// TIA Portal V19 export
FUNCTION "PREMIXING" : Void   // FC19, LAD
{ S7_Optimized_Access := 'TRUE' }
// stored: SetENOAutomatically false
   VAR_TEMP   // added for the SCL form of the ladder/FBD networks
      _w1 : Bool;
   END_VAR
BEGIN

REGION Network 2: START MFG PROCESS
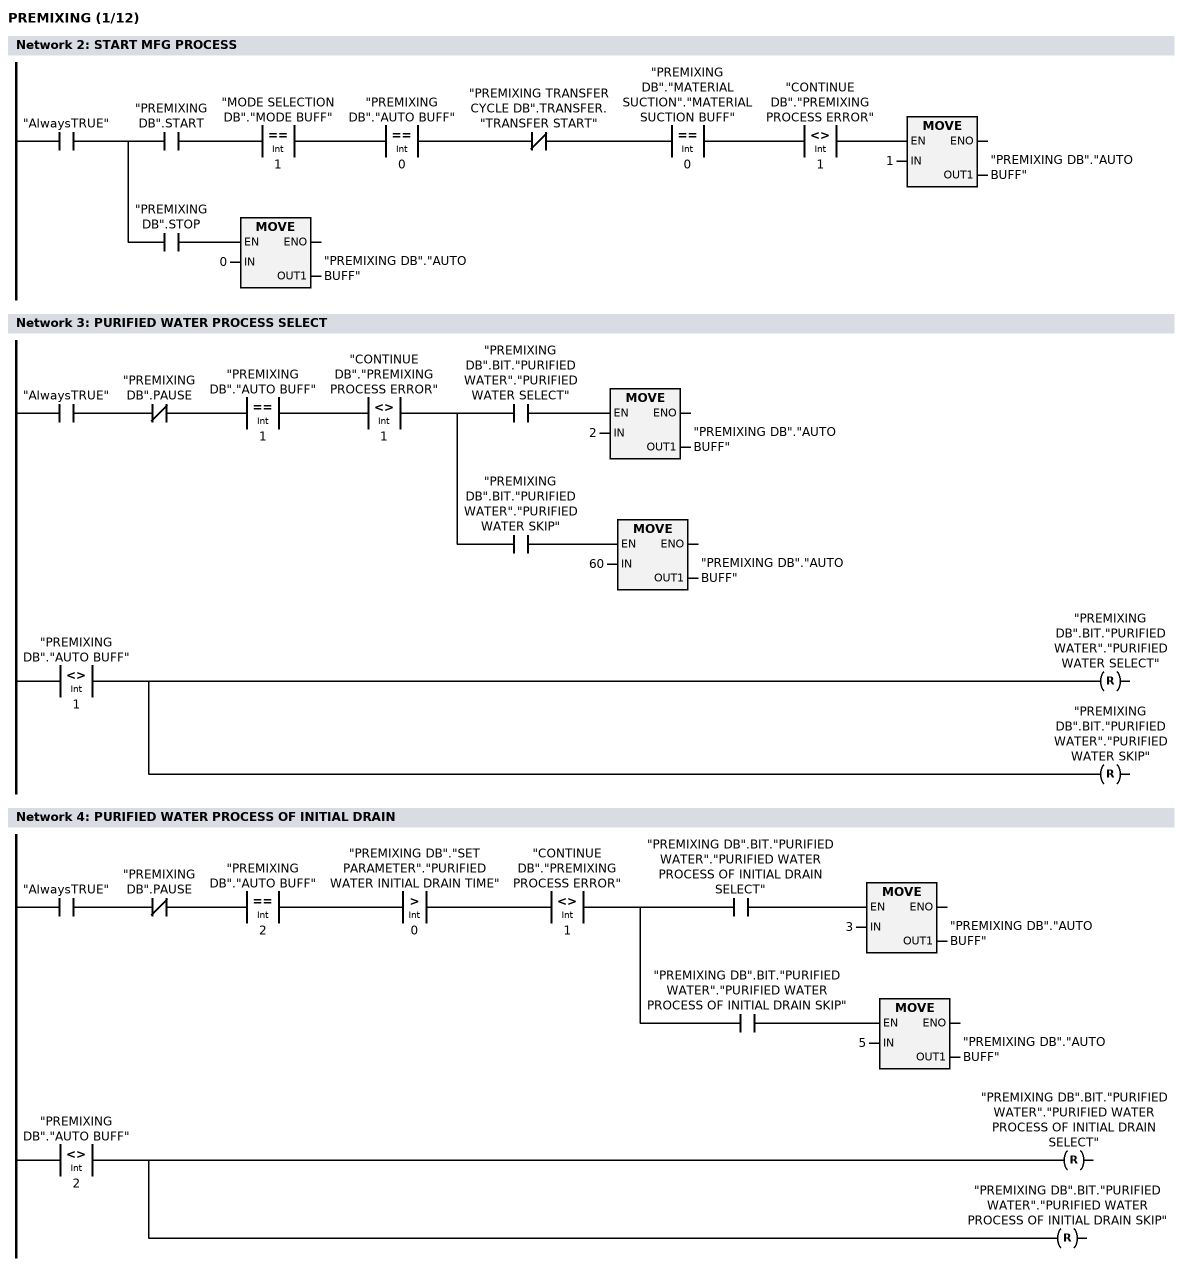
   RUNG wire#powerrail
      Contact( "AlwaysTRUE" )
      wire#w1
      Contact( "PREMIXING DB".START )
      { S7_Templates := "SrcType := Int" } EQ_Contact(in1 := "MODE SELECTION DB"."MODE BUFF", in2 := 1)
      { S7_Templates := "SrcType := Int" } EQ_Contact(in1 := "PREMIXING DB"."AUTO BUFF", in2 := 0)
      I_Contact( "PREMIXING TRANSFER CYCLE DB".TRANSFER."TRANSFER START" )
      { S7_Templates := "SrcType := Int" } EQ_Contact(in1 := "PREMIXING DB"."MATERIAL SUCTION"."MATERIAL SUCTION BUFF", in2 := 0)
      { S7_Templates := "SrcType := Int" } NE_Contact(in1 := "CONTINUE DB"."PREMIXING PROCESS ERROR", in2 := 1)
      Move(in := 1, out1 => "PREMIXING DB"."AUTO BUFF")
   END_RUNG
   RUNG wire#w1
      Contact( "PREMIXING DB".STOP )
      Move(in := 0, out1 => "PREMIXING DB"."AUTO BUFF")
   END_RUNG
   // the same network as SCL:
   IF "AlwaysTRUE" AND "PREMIXING DB".START AND ("MODE SELECTION DB"."MODE BUFF" = 1) AND ("PREMIXING DB"."AUTO BUFF" = 0) AND NOT "PREMIXING TRANSFER CYCLE DB".TRANSFER."TRANSFER START" AND ("PREMIXING DB"."MATERIAL SUCTION"."MATERIAL SUCTION BUFF" = 0) AND ("CONTINUE DB"."PREMIXING PROCESS ERROR" <> 1) THEN
       "PREMIXING DB"."AUTO BUFF" := 1;
   END_IF;
   IF "AlwaysTRUE" AND "PREMIXING DB".STOP THEN "PREMIXING DB"."AUTO BUFF" := 0; END_IF;
END_REGION

REGION Network 3: PURIFIED WATER PROCESS SELECT
   RUNG wire#powerrail
      Contact( "AlwaysTRUE" )
      I_Contact( "PREMIXING DB".PAUSE )
      { S7_Templates := "SrcType := Int" } EQ_Contact(in1 := "PREMIXING DB"."AUTO BUFF", in2 := 1)
      { S7_Templates := "SrcType := Int" } NE_Contact(in1 := "CONTINUE DB"."PREMIXING PROCESS ERROR", in2 := 1)
      wire#w1
      Contact( "PREMIXING DB".BIT."PURIFIED WATER"."PURIFIED WATER SELECT" )
      Move(in := 2, out1 => "PREMIXING DB"."AUTO BUFF")
   END_RUNG
   RUNG wire#w1
      Contact( "PREMIXING DB".BIT."PURIFIED WATER"."PURIFIED WATER SKIP" )
      Move(in := 60, out1 => "PREMIXING DB"."AUTO BUFF")
   END_RUNG
   RUNG wire#powerrail
      { S7_Templates := "SrcType := Int" } NE_Contact(in1 := "PREMIXING DB"."AUTO BUFF", in2 := 1)
      wire#w2
      R_Coil( "PREMIXING DB".BIT."PURIFIED WATER"."PURIFIED WATER SELECT" )
   END_RUNG
   RUNG wire#w2
      R_Coil( "PREMIXING DB".BIT."PURIFIED WATER"."PURIFIED WATER SKIP" )
   END_RUNG
   // the same network as SCL:
   #_w1 := "AlwaysTRUE" AND NOT "PREMIXING DB".PAUSE AND ("PREMIXING DB"."AUTO BUFF" = 1) AND ("CONTINUE DB"."PREMIXING PROCESS ERROR" <> 1);
   IF #_w1 AND "PREMIXING DB".BIT."PURIFIED WATER"."PURIFIED WATER SELECT" THEN
       "PREMIXING DB"."AUTO BUFF" := 2;
   END_IF;
   IF #_w1 AND "PREMIXING DB".BIT."PURIFIED WATER"."PURIFIED WATER SKIP" THEN
       "PREMIXING DB"."AUTO BUFF" := 60;
   END_IF;
   IF "PREMIXING DB"."AUTO BUFF" <> 1 THEN
       "PREMIXING DB".BIT."PURIFIED WATER"."PURIFIED WATER SELECT" := FALSE;
       "PREMIXING DB".BIT."PURIFIED WATER"."PURIFIED WATER SKIP" := FALSE;
   END_IF;
END_REGION

REGION Network 4: PURIFIED WATER PROCESS OF INITIAL DRAIN
   RUNG wire#powerrail
      Contact( "AlwaysTRUE" )
      I_Contact( "PREMIXING DB".PAUSE )
      { S7_Templates := "SrcType := Int" } EQ_Contact(in1 := "PREMIXING DB"."AUTO BUFF", in2 := 2)
      { S7_Templates := "SrcType := Int" } GT_Contact(in1 := "PREMIXING DB"."SET PARAMETER"."PURIFIED WATER INITIAL DRAIN TIME", in2 := 0)
      { S7_Templates := "SrcType := Int" } NE_Contact(in1 := "CONTINUE DB"."PREMIXING PROCESS ERROR", in2 := 1)
      wire#w1
      Contact( "PREMIXING DB".BIT."PURIFIED WATER"."PURIFIED WATER PROCESS OF INITIAL DRAIN SELECT" )
      Move(in := 3, out1 => "PREMIXING DB"."AUTO BUFF")
   END_RUNG
   RUNG wire#w1
      Contact( "PREMIXING DB".BIT."PURIFIED WATER"."PURIFIED WATER PROCESS OF INITIAL DRAIN SKIP" )
      Move(in := 5, out1 => "PREMIXING DB"."AUTO BUFF")
   END_RUNG
   RUNG wire#powerrail
      { S7_Templates := "SrcType := Int" } NE_Contact(in1 := "PREMIXING DB"."AUTO BUFF", in2 := 2)
      wire#w2
      R_Coil( "PREMIXING DB".BIT."PURIFIED WATER"."PURIFIED WATER PROCESS OF INITIAL DRAIN SELECT" )
   END_RUNG
   RUNG wire#w2
      R_Coil( "PREMIXING DB".BIT."PURIFIED WATER"."PURIFIED WATER PROCESS OF INITIAL DRAIN SKIP" )
   END_RUNG
   // the same network as SCL:
   #_w1 := "AlwaysTRUE" AND NOT "PREMIXING DB".PAUSE AND ("PREMIXING DB"."AUTO BUFF" = 2) AND ("PREMIXING DB"."SET PARAMETER"."PURIFIED WATER INITIAL DRAIN TIME" > 0) AND ("CONTINUE DB"."PREMIXING PROCESS ERROR" <> 1);
   IF #_w1 AND "PREMIXING DB".BIT."PURIFIED WATER"."PURIFIED WATER PROCESS OF INITIAL DRAIN SELECT" THEN
       "PREMIXING DB"."AUTO BUFF" := 3;
   END_IF;
   IF #_w1 AND "PREMIXING DB".BIT."PURIFIED WATER"."PURIFIED WATER PROCESS OF INITIAL DRAIN SKIP" THEN
       "PREMIXING DB"."AUTO BUFF" := 5;
   END_IF;
   IF "PREMIXING DB"."AUTO BUFF" <> 2 THEN
       "PREMIXING DB".BIT."PURIFIED WATER"."PURIFIED WATER PROCESS OF INITIAL DRAIN SELECT" := FALSE;
       "PREMIXING DB".BIT."PURIFIED WATER"."PURIFIED WATER PROCESS OF INITIAL DRAIN SKIP" := FALSE;
   END_IF;
END_REGION

REGION Network 5: TIMER
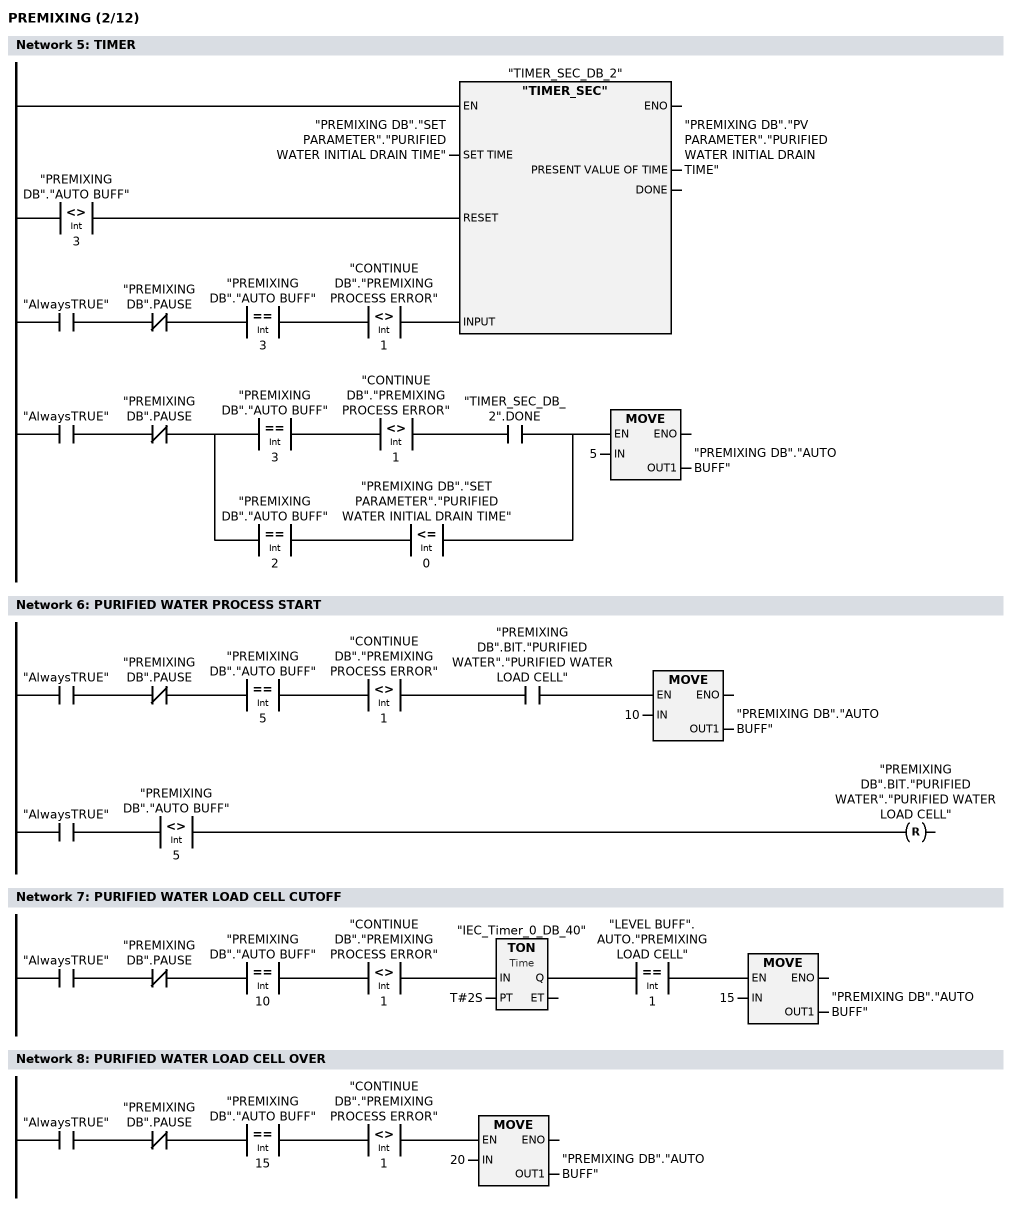
   RUNG wire#powerrail
      "TIMER_SEC_DB_2"(RESET := wire#w1, INPUT := wire#w2, "SET TIME" := "PREMIXING DB"."SET PARAMETER"."PURIFIED WATER INITIAL DRAIN TIME", "PRESENT VALUE OF TIME" => "PREMIXING DB"."PV PARAMETER"."PURIFIED WATER INITIAL DRAIN TIME", DONE =>)
   END_RUNG
   RUNG wire#powerrail
      { S7_Templates := "SrcType := Int" } NE_Contact(in1 := "PREMIXING DB"."AUTO BUFF", in2 := 3)
   END_RUNG wire#w1
   RUNG wire#powerrail
      Contact( "AlwaysTRUE" )
      I_Contact( "PREMIXING DB".PAUSE )
      { S7_Templates := "SrcType := Int" } EQ_Contact(in1 := "PREMIXING DB"."AUTO BUFF", in2 := 3)
      { S7_Templates := "SrcType := Int" } NE_Contact(in1 := "CONTINUE DB"."PREMIXING PROCESS ERROR", in2 := 1)
   END_RUNG wire#w2
   RUNG wire#powerrail
      Contact( "AlwaysTRUE" )
      I_Contact( "PREMIXING DB".PAUSE )
      wire#w3
      { S7_Templates := "SrcType := Int" } EQ_Contact(in1 := "PREMIXING DB"."AUTO BUFF", in2 := 3)
      { S7_Templates := "SrcType := Int" } NE_Contact(in1 := "CONTINUE DB"."PREMIXING PROCESS ERROR", in2 := 1)
      Contact( "TIMER_SEC_DB_2".DONE )
      wire#w4
      Move(in := 5, out1 => "PREMIXING DB"."AUTO BUFF")
   END_RUNG
   RUNG wire#w3
      { S7_Templates := "SrcType := Int" } EQ_Contact(in1 := "PREMIXING DB"."AUTO BUFF", in2 := 2)
      { S7_Templates := "SrcType := Int" } LE_Contact(in1 := "PREMIXING DB"."SET PARAMETER"."PURIFIED WATER INITIAL DRAIN TIME", in2 := 0)
   END_RUNG wire#w4
   // the same network as SCL:
   "TIMER_SEC_DB_2"("SET TIME" := "PREMIXING DB"."SET PARAMETER"."PURIFIED WATER INITIAL DRAIN TIME",   // "TIMER_SEC"
                    RESET := "PREMIXING DB"."AUTO BUFF" <> 3,
                    INPUT := "AlwaysTRUE" AND NOT "PREMIXING DB".PAUSE AND ("PREMIXING DB"."AUTO BUFF" = 3) AND ("CONTINUE DB"."PREMIXING PROCESS ERROR" <> 1),
                    "PRESENT VALUE OF TIME" => "PREMIXING DB"."PV PARAMETER"."PURIFIED WATER INITIAL DRAIN TIME");
   IF "AlwaysTRUE" AND NOT "PREMIXING DB".PAUSE AND ((("PREMIXING DB"."AUTO BUFF" = 3) AND ("CONTINUE DB"."PREMIXING PROCESS ERROR" <> 1) AND "TIMER_SEC_DB_2".DONE) OR (("PREMIXING DB"."AUTO BUFF" = 2) AND ("PREMIXING DB"."SET PARAMETER"."PURIFIED WATER INITIAL DRAIN TIME" <= 0))) THEN
       "PREMIXING DB"."AUTO BUFF" := 5;
   END_IF;
END_REGION

REGION Network 6: PURIFIED WATER PROCESS START
   RUNG wire#powerrail
      Contact( "AlwaysTRUE" )
      I_Contact( "PREMIXING DB".PAUSE )
      { S7_Templates := "SrcType := Int" } EQ_Contact(in1 := "PREMIXING DB"."AUTO BUFF", in2 := 5)
      { S7_Templates := "SrcType := Int" } NE_Contact(in1 := "CONTINUE DB"."PREMIXING PROCESS ERROR", in2 := 1)
      Contact( "PREMIXING DB".BIT."PURIFIED WATER"."PURIFIED WATER LOAD CELL" )
      Move(in := 10, out1 => "PREMIXING DB"."AUTO BUFF")
   END_RUNG
   RUNG wire#powerrail
      Contact( "AlwaysTRUE" )
      { S7_Templates := "SrcType := Int" } NE_Contact(in1 := "PREMIXING DB"."AUTO BUFF", in2 := 5)
      R_Coil( "PREMIXING DB".BIT."PURIFIED WATER"."PURIFIED WATER LOAD CELL" )
   END_RUNG
   // the same network as SCL:
   IF "AlwaysTRUE" AND NOT "PREMIXING DB".PAUSE AND ("PREMIXING DB"."AUTO BUFF" = 5) AND ("CONTINUE DB"."PREMIXING PROCESS ERROR" <> 1) AND "PREMIXING DB".BIT."PURIFIED WATER"."PURIFIED WATER LOAD CELL" THEN
       "PREMIXING DB"."AUTO BUFF" := 10;
   END_IF;
   IF "AlwaysTRUE" AND ("PREMIXING DB"."AUTO BUFF" <> 5) THEN
       "PREMIXING DB".BIT."PURIFIED WATER"."PURIFIED WATER LOAD CELL" := FALSE;
   END_IF;
END_REGION

REGION Network 7: PURIFIED WATER LOAD CELL CUTOFF
   RUNG wire#powerrail
      Contact( "AlwaysTRUE" )
      I_Contact( "PREMIXING DB".PAUSE )
      { S7_Templates := "SrcType := Int" } EQ_Contact(in1 := "PREMIXING DB"."AUTO BUFF", in2 := 10)
      { S7_Templates := "SrcType := Int" } NE_Contact(in1 := "CONTINUE DB"."PREMIXING PROCESS ERROR", in2 := 1)
      { S7_Templates := "time_type := Time" } "IEC_Timer_0_DB_40".TON(pt := T#2S, et =>)
      { S7_Templates := "SrcType := Int" } EQ_Contact(in1 := "LEVEL BUFF".AUTO."PREMIXING LOAD CELL", in2 := 1)
      Move(in := 15, out1 => "PREMIXING DB"."AUTO BUFF")
   END_RUNG
   // the same network as SCL:
   "IEC_Timer_0_DB_40".TON(IN := "AlwaysTRUE" AND NOT "PREMIXING DB".PAUSE AND ("PREMIXING DB"."AUTO BUFF" = 10) AND ("CONTINUE DB"."PREMIXING PROCESS ERROR" <> 1),
                           PT := T#2S);
   IF "IEC_Timer_0_DB_40".Q AND ("LEVEL BUFF".AUTO."PREMIXING LOAD CELL" = 1) THEN
       "PREMIXING DB"."AUTO BUFF" := 15;
   END_IF;
END_REGION

REGION Network 8: PURIFIED WATER LOAD CELL OVER
   RUNG wire#powerrail
      Contact( "AlwaysTRUE" )
      I_Contact( "PREMIXING DB".PAUSE )
      { S7_Templates := "SrcType := Int" } EQ_Contact(in1 := "PREMIXING DB"."AUTO BUFF", in2 := 15)
      { S7_Templates := "SrcType := Int" } NE_Contact(in1 := "CONTINUE DB"."PREMIXING PROCESS ERROR", in2 := 1)
      Move(in := 20, out1 => "PREMIXING DB"."AUTO BUFF")
   END_RUNG
   // the same network as SCL:
   IF "AlwaysTRUE" AND NOT "PREMIXING DB".PAUSE AND ("PREMIXING DB"."AUTO BUFF" = 15) AND ("CONTINUE DB"."PREMIXING PROCESS ERROR" <> 1) THEN
       "PREMIXING DB"."AUTO BUFF" := 20;
   END_IF;
END_REGION

REGION Network 9: PURIFIED WATER HEATING OR COOLING SEL
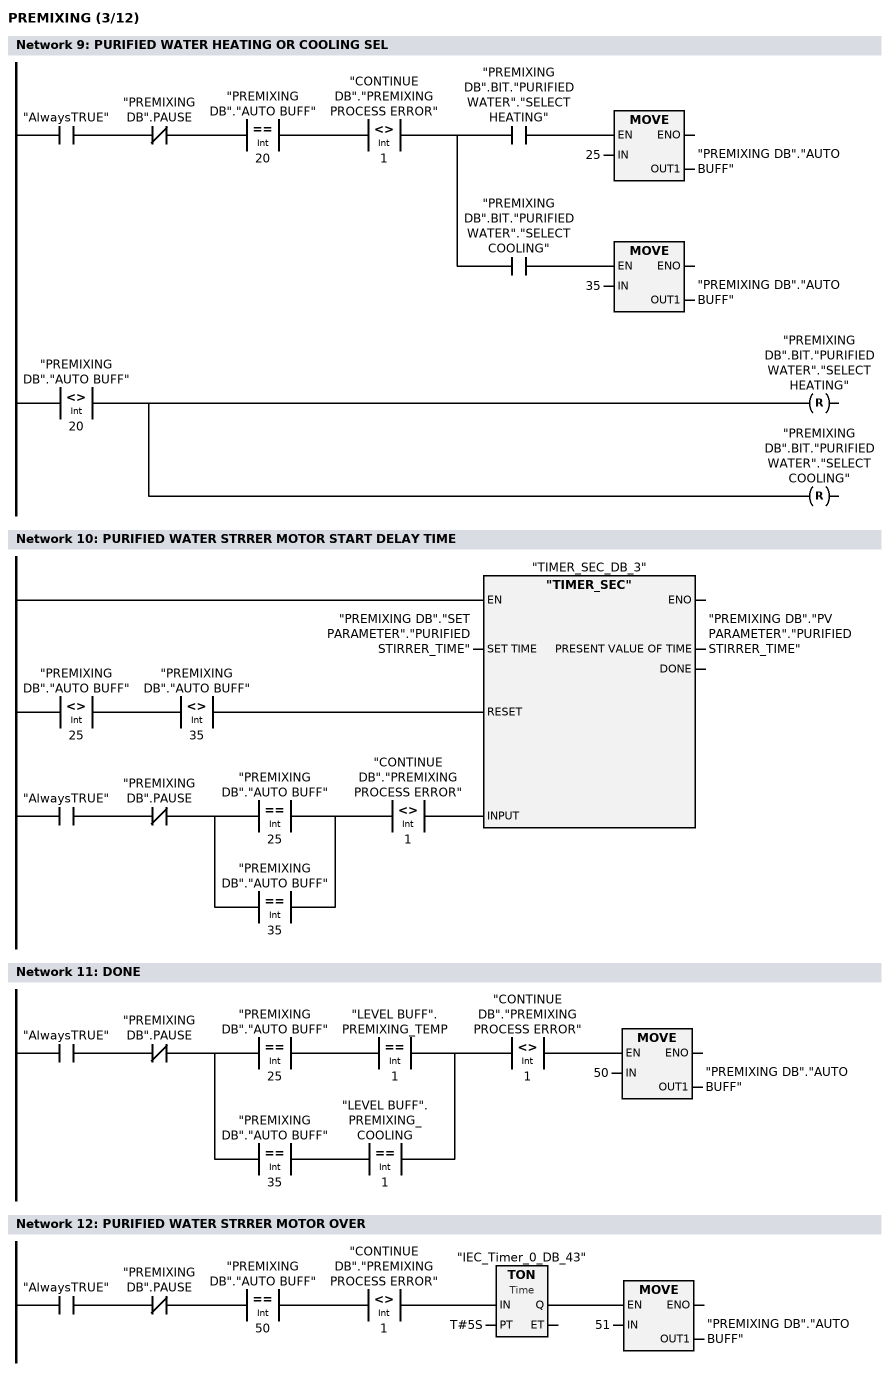
   RUNG wire#powerrail
      Contact( "AlwaysTRUE" )
      I_Contact( "PREMIXING DB".PAUSE )
      { S7_Templates := "SrcType := Int" } EQ_Contact(in1 := "PREMIXING DB"."AUTO BUFF", in2 := 20)
      { S7_Templates := "SrcType := Int" } NE_Contact(in1 := "CONTINUE DB"."PREMIXING PROCESS ERROR", in2 := 1)
      wire#w1
      Contact( "PREMIXING DB".BIT."PURIFIED WATER"."SELECT HEATING" )
      Move(in := 25, out1 => "PREMIXING DB"."AUTO BUFF")
   END_RUNG
   RUNG wire#w1
      Contact( "PREMIXING DB".BIT."PURIFIED WATER"."SELECT COOLING" )
      Move(in := 35, out1 => "PREMIXING DB"."AUTO BUFF")
   END_RUNG
   RUNG wire#powerrail
      { S7_Templates := "SrcType := Int" } NE_Contact(in1 := "PREMIXING DB"."AUTO BUFF", in2 := 20)
      wire#w2
      R_Coil( "PREMIXING DB".BIT."PURIFIED WATER"."SELECT HEATING" )
   END_RUNG
   RUNG wire#w2
      R_Coil( "PREMIXING DB".BIT."PURIFIED WATER"."SELECT COOLING" )
   END_RUNG
   // the same network as SCL:
   #_w1 := "AlwaysTRUE" AND NOT "PREMIXING DB".PAUSE AND ("PREMIXING DB"."AUTO BUFF" = 20) AND ("CONTINUE DB"."PREMIXING PROCESS ERROR" <> 1);
   IF #_w1 AND "PREMIXING DB".BIT."PURIFIED WATER"."SELECT HEATING" THEN
       "PREMIXING DB"."AUTO BUFF" := 25;
   END_IF;
   IF #_w1 AND "PREMIXING DB".BIT."PURIFIED WATER"."SELECT COOLING" THEN
       "PREMIXING DB"."AUTO BUFF" := 35;
   END_IF;
   IF "PREMIXING DB"."AUTO BUFF" <> 20 THEN
       "PREMIXING DB".BIT."PURIFIED WATER"."SELECT HEATING" := FALSE;
       "PREMIXING DB".BIT."PURIFIED WATER"."SELECT COOLING" := FALSE;
   END_IF;
END_REGION

REGION Network 10: PURIFIED WATER STRRER MOTOR START DELAY TIME
   RUNG wire#powerrail
      "TIMER_SEC_DB_3"(RESET := wire#w1, INPUT := wire#w4, "SET TIME" := "PREMIXING DB"."SET PARAMETER"."PURIFIED STIRRER_TIME", "PRESENT VALUE OF TIME" => "PREMIXING DB"."PV PARAMETER"."PURIFIED STIRRER_TIME", DONE =>)
   END_RUNG
   RUNG wire#powerrail
      { S7_Templates := "SrcType := Int" } NE_Contact(in1 := "PREMIXING DB"."AUTO BUFF", in2 := 25)
      { S7_Templates := "SrcType := Int" } NE_Contact(in1 := "PREMIXING DB"."AUTO BUFF", in2 := 35)
   END_RUNG wire#w1
   RUNG wire#powerrail
      Contact( "AlwaysTRUE" )
      I_Contact( "PREMIXING DB".PAUSE )
      wire#w2
      { S7_Templates := "SrcType := Int" } EQ_Contact(in1 := "PREMIXING DB"."AUTO BUFF", in2 := 25)
      wire#w3
      { S7_Templates := "SrcType := Int" } NE_Contact(in1 := "CONTINUE DB"."PREMIXING PROCESS ERROR", in2 := 1)
   END_RUNG wire#w4
   RUNG wire#w2
      { S7_Templates := "SrcType := Int" } EQ_Contact(in1 := "PREMIXING DB"."AUTO BUFF", in2 := 35)
   END_RUNG wire#w3
   // the same network as SCL:
   "TIMER_SEC_DB_3"("SET TIME" := "PREMIXING DB"."SET PARAMETER"."PURIFIED STIRRER_TIME",   // "TIMER_SEC"
                    RESET := ("PREMIXING DB"."AUTO BUFF" <> 25) AND ("PREMIXING DB"."AUTO BUFF" <> 35),
                    INPUT := "AlwaysTRUE" AND NOT "PREMIXING DB".PAUSE AND (("PREMIXING DB"."AUTO BUFF" = 25) OR ("PREMIXING DB"."AUTO BUFF" = 35)) AND ("CONTINUE DB"."PREMIXING PROCESS ERROR" <> 1),
                    "PRESENT VALUE OF TIME" => "PREMIXING DB"."PV PARAMETER"."PURIFIED STIRRER_TIME");
END_REGION

REGION Network 11: DONE
   RUNG wire#powerrail
      Contact( "AlwaysTRUE" )
      I_Contact( "PREMIXING DB".PAUSE )
      wire#w1
      { S7_Templates := "SrcType := Int" } EQ_Contact(in1 := "PREMIXING DB"."AUTO BUFF", in2 := 25)
      { S7_Templates := "SrcType := Int" } EQ_Contact(in1 := "LEVEL BUFF".PREMIXING_TEMP, in2 := 1)
      wire#w2
      { S7_Templates := "SrcType := Int" } NE_Contact(in1 := "CONTINUE DB"."PREMIXING PROCESS ERROR", in2 := 1)
      Move(in := 50, out1 => "PREMIXING DB"."AUTO BUFF")
   END_RUNG
   RUNG wire#w1
      { S7_Templates := "SrcType := Int" } EQ_Contact(in1 := "PREMIXING DB"."AUTO BUFF", in2 := 35)
      { S7_Templates := "SrcType := Int" } EQ_Contact(in1 := "LEVEL BUFF".PREMIXING_COOLING, in2 := 1)
   END_RUNG wire#w2
   // the same network as SCL:
   IF "AlwaysTRUE" AND NOT "PREMIXING DB".PAUSE AND ((("PREMIXING DB"."AUTO BUFF" = 25) AND ("LEVEL BUFF".PREMIXING_TEMP = 1)) OR (("PREMIXING DB"."AUTO BUFF" = 35) AND ("LEVEL BUFF".PREMIXING_COOLING = 1))) AND ("CONTINUE DB"."PREMIXING PROCESS ERROR" <> 1) THEN
       "PREMIXING DB"."AUTO BUFF" := 50;
   END_IF;
END_REGION

REGION Network 12: PURIFIED WATER STRRER MOTOR OVER
   RUNG wire#powerrail
      Contact( "AlwaysTRUE" )
      I_Contact( "PREMIXING DB".PAUSE )
      { S7_Templates := "SrcType := Int" } EQ_Contact(in1 := "PREMIXING DB"."AUTO BUFF", in2 := 50)
      { S7_Templates := "SrcType := Int" } NE_Contact(in1 := "CONTINUE DB"."PREMIXING PROCESS ERROR", in2 := 1)
      { S7_Templates := "time_type := Time" } "IEC_Timer_0_DB_43".TON(pt := T#5S, et =>)
      Move(in := 51, out1 => "PREMIXING DB"."AUTO BUFF")
   END_RUNG
   // the same network as SCL:
   "IEC_Timer_0_DB_43".TON(IN := "AlwaysTRUE" AND NOT "PREMIXING DB".PAUSE AND ("PREMIXING DB"."AUTO BUFF" = 50) AND ("CONTINUE DB"."PREMIXING PROCESS ERROR" <> 1),
                           PT := T#5S);
   IF "IEC_Timer_0_DB_43".Q THEN "PREMIXING DB"."AUTO BUFF" := 51; END_IF;
END_REGION

REGION Network 13: PURIFIED WATER PROCESS OF JACKET DRAIN
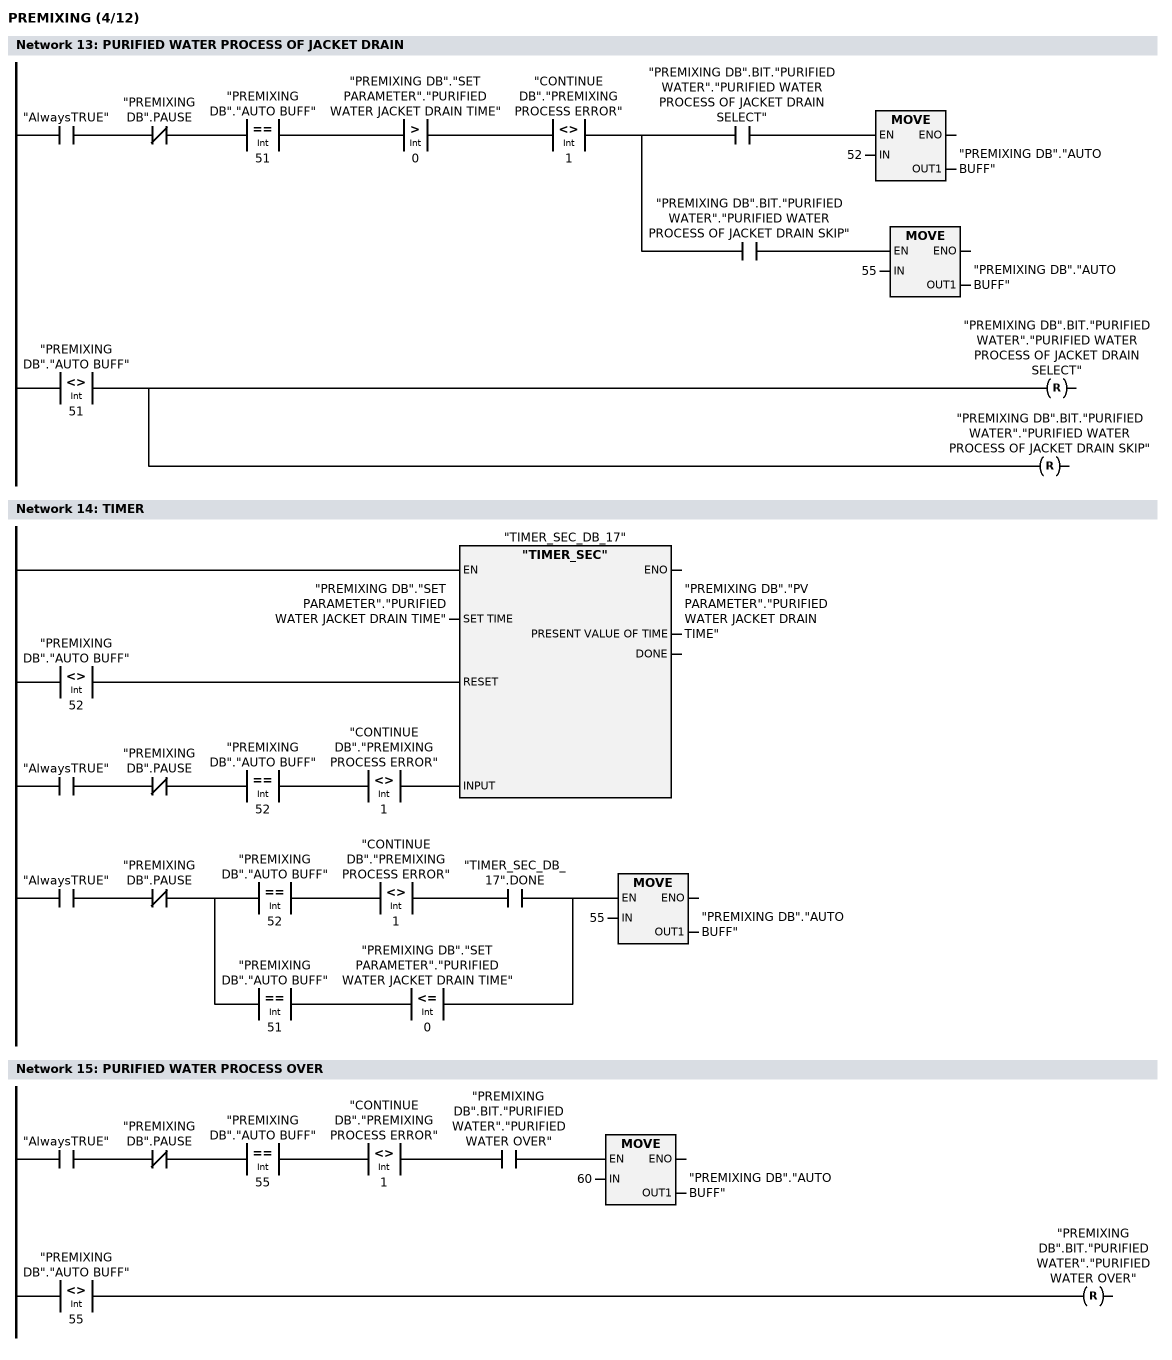
   RUNG wire#powerrail
      Contact( "AlwaysTRUE" )
      I_Contact( "PREMIXING DB".PAUSE )
      { S7_Templates := "SrcType := Int" } EQ_Contact(in1 := "PREMIXING DB"."AUTO BUFF", in2 := 51)
      { S7_Templates := "SrcType := Int" } GT_Contact(in1 := "PREMIXING DB"."SET PARAMETER"."PURIFIED WATER JACKET DRAIN TIME", in2 := 0)
      { S7_Templates := "SrcType := Int" } NE_Contact(in1 := "CONTINUE DB"."PREMIXING PROCESS ERROR", in2 := 1)
      wire#w1
      Contact( "PREMIXING DB".BIT."PURIFIED WATER"."PURIFIED WATER PROCESS OF JACKET DRAIN SELECT" )
      Move(in := 52, out1 => "PREMIXING DB"."AUTO BUFF")
   END_RUNG
   RUNG wire#w1
      Contact( "PREMIXING DB".BIT."PURIFIED WATER"."PURIFIED WATER PROCESS OF JACKET DRAIN SKIP" )
      Move(in := 55, out1 => "PREMIXING DB"."AUTO BUFF")
   END_RUNG
   RUNG wire#powerrail
      { S7_Templates := "SrcType := Int" } NE_Contact(in1 := "PREMIXING DB"."AUTO BUFF", in2 := 51)
      wire#w2
      R_Coil( "PREMIXING DB".BIT."PURIFIED WATER"."PURIFIED WATER PROCESS OF JACKET DRAIN SELECT" )
   END_RUNG
   RUNG wire#w2
      R_Coil( "PREMIXING DB".BIT."PURIFIED WATER"."PURIFIED WATER PROCESS OF JACKET DRAIN SKIP" )
   END_RUNG
   // the same network as SCL:
   #_w1 := "AlwaysTRUE" AND NOT "PREMIXING DB".PAUSE AND ("PREMIXING DB"."AUTO BUFF" = 51) AND ("PREMIXING DB"."SET PARAMETER"."PURIFIED WATER JACKET DRAIN TIME" > 0) AND ("CONTINUE DB"."PREMIXING PROCESS ERROR" <> 1);
   IF #_w1 AND "PREMIXING DB".BIT."PURIFIED WATER"."PURIFIED WATER PROCESS OF JACKET DRAIN SELECT" THEN
       "PREMIXING DB"."AUTO BUFF" := 52;
   END_IF;
   IF #_w1 AND "PREMIXING DB".BIT."PURIFIED WATER"."PURIFIED WATER PROCESS OF JACKET DRAIN SKIP" THEN
       "PREMIXING DB"."AUTO BUFF" := 55;
   END_IF;
   IF "PREMIXING DB"."AUTO BUFF" <> 51 THEN
       "PREMIXING DB".BIT."PURIFIED WATER"."PURIFIED WATER PROCESS OF JACKET DRAIN SELECT" := FALSE;
       "PREMIXING DB".BIT."PURIFIED WATER"."PURIFIED WATER PROCESS OF JACKET DRAIN SKIP" := FALSE;
   END_IF;
END_REGION

REGION Network 14: TIMER
   RUNG wire#powerrail
      "TIMER_SEC_DB_17"(RESET := wire#w1, INPUT := wire#w2, "SET TIME" := "PREMIXING DB"."SET PARAMETER"."PURIFIED WATER JACKET DRAIN TIME", "PRESENT VALUE OF TIME" => "PREMIXING DB"."PV PARAMETER"."PURIFIED WATER JACKET DRAIN TIME", DONE =>)
   END_RUNG
   RUNG wire#powerrail
      { S7_Templates := "SrcType := Int" } NE_Contact(in1 := "PREMIXING DB"."AUTO BUFF", in2 := 52)
   END_RUNG wire#w1
   RUNG wire#powerrail
      Contact( "AlwaysTRUE" )
      I_Contact( "PREMIXING DB".PAUSE )
      { S7_Templates := "SrcType := Int" } EQ_Contact(in1 := "PREMIXING DB"."AUTO BUFF", in2 := 52)
      { S7_Templates := "SrcType := Int" } NE_Contact(in1 := "CONTINUE DB"."PREMIXING PROCESS ERROR", in2 := 1)
   END_RUNG wire#w2
   RUNG wire#powerrail
      Contact( "AlwaysTRUE" )
      I_Contact( "PREMIXING DB".PAUSE )
      wire#w3
      { S7_Templates := "SrcType := Int" } EQ_Contact(in1 := "PREMIXING DB"."AUTO BUFF", in2 := 52)
      { S7_Templates := "SrcType := Int" } NE_Contact(in1 := "CONTINUE DB"."PREMIXING PROCESS ERROR", in2 := 1)
      Contact( "TIMER_SEC_DB_17".DONE )
      wire#w4
      Move(in := 55, out1 => "PREMIXING DB"."AUTO BUFF")
   END_RUNG
   RUNG wire#w3
      { S7_Templates := "SrcType := Int" } EQ_Contact(in1 := "PREMIXING DB"."AUTO BUFF", in2 := 51)
      { S7_Templates := "SrcType := Int" } LE_Contact(in1 := "PREMIXING DB"."SET PARAMETER"."PURIFIED WATER JACKET DRAIN TIME", in2 := 0)
   END_RUNG wire#w4
   // the same network as SCL:
   "TIMER_SEC_DB_17"("SET TIME" := "PREMIXING DB"."SET PARAMETER"."PURIFIED WATER JACKET DRAIN TIME",   // "TIMER_SEC"
                     RESET := "PREMIXING DB"."AUTO BUFF" <> 52,
                     INPUT := "AlwaysTRUE" AND NOT "PREMIXING DB".PAUSE AND ("PREMIXING DB"."AUTO BUFF" = 52) AND ("CONTINUE DB"."PREMIXING PROCESS ERROR" <> 1),
                     "PRESENT VALUE OF TIME" => "PREMIXING DB"."PV PARAMETER"."PURIFIED WATER JACKET DRAIN TIME");
   IF "AlwaysTRUE" AND NOT "PREMIXING DB".PAUSE AND ((("PREMIXING DB"."AUTO BUFF" = 52) AND ("CONTINUE DB"."PREMIXING PROCESS ERROR" <> 1) AND "TIMER_SEC_DB_17".DONE) OR (("PREMIXING DB"."AUTO BUFF" = 51) AND ("PREMIXING DB"."SET PARAMETER"."PURIFIED WATER JACKET DRAIN TIME" <= 0))) THEN
       "PREMIXING DB"."AUTO BUFF" := 55;
   END_IF;
END_REGION

REGION Network 15: PURIFIED WATER PROCESS OVER
   RUNG wire#powerrail
      Contact( "AlwaysTRUE" )
      I_Contact( "PREMIXING DB".PAUSE )
      { S7_Templates := "SrcType := Int" } EQ_Contact(in1 := "PREMIXING DB"."AUTO BUFF", in2 := 55)
      { S7_Templates := "SrcType := Int" } NE_Contact(in1 := "CONTINUE DB"."PREMIXING PROCESS ERROR", in2 := 1)
      Contact( "PREMIXING DB".BIT."PURIFIED WATER"."PURIFIED WATER OVER" )
      Move(in := 60, out1 => "PREMIXING DB"."AUTO BUFF")
   END_RUNG
   RUNG wire#powerrail
      { S7_Templates := "SrcType := Int" } NE_Contact(in1 := "PREMIXING DB"."AUTO BUFF", in2 := 55)
      R_Coil( "PREMIXING DB".BIT."PURIFIED WATER"."PURIFIED WATER OVER" )
   END_RUNG
   // the same network as SCL:
   IF "AlwaysTRUE" AND NOT "PREMIXING DB".PAUSE AND ("PREMIXING DB"."AUTO BUFF" = 55) AND ("CONTINUE DB"."PREMIXING PROCESS ERROR" <> 1) AND "PREMIXING DB".BIT."PURIFIED WATER"."PURIFIED WATER OVER" THEN
       "PREMIXING DB"."AUTO BUFF" := 60;
   END_IF;
   IF "PREMIXING DB"."AUTO BUFF" <> 55 THEN
       "PREMIXING DB".BIT."PURIFIED WATER"."PURIFIED WATER OVER" := FALSE;
   END_IF;
END_REGION

REGION Network 17: MATERIAL ADDITION PROCESS SELECT
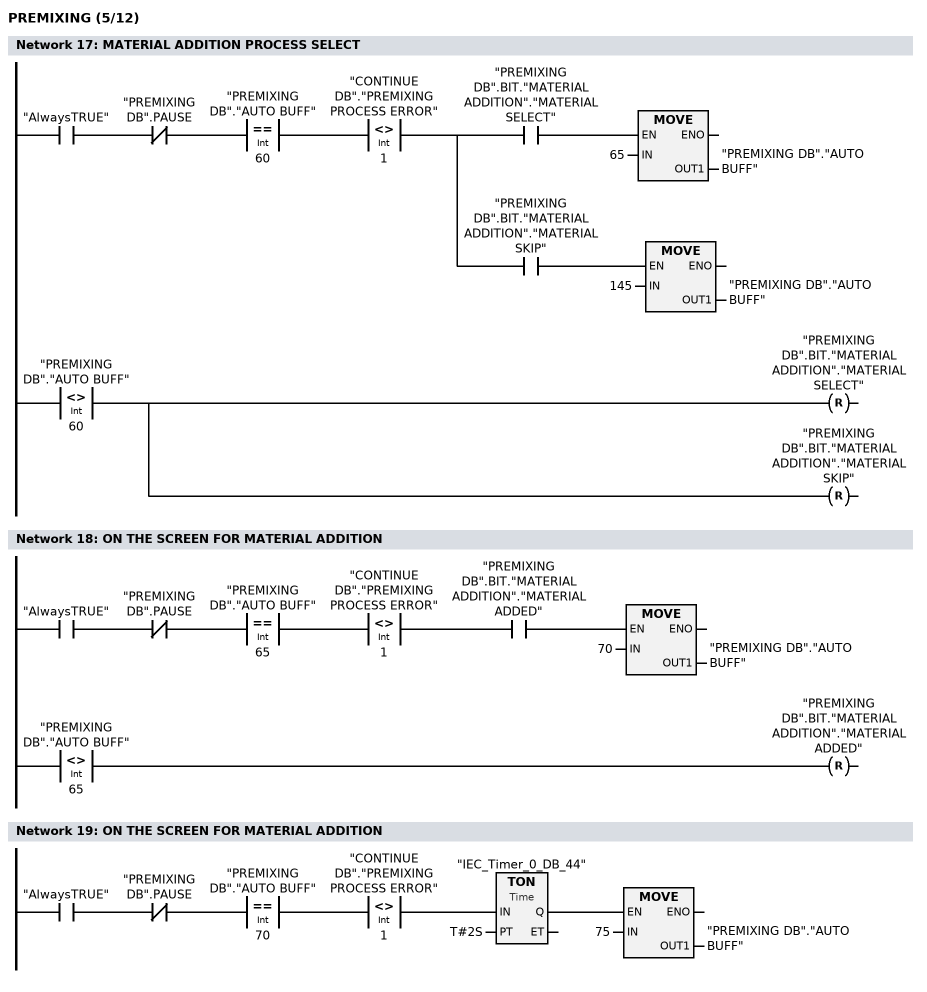
   RUNG wire#powerrail
      Contact( "AlwaysTRUE" )
      I_Contact( "PREMIXING DB".PAUSE )
      { S7_Templates := "SrcType := Int" } EQ_Contact(in1 := "PREMIXING DB"."AUTO BUFF", in2 := 60)
      { S7_Templates := "SrcType := Int" } NE_Contact(in1 := "CONTINUE DB"."PREMIXING PROCESS ERROR", in2 := 1)
      wire#w1
      Contact( "PREMIXING DB".BIT."MATERIAL ADDITION"."MATERIAL SELECT" )
      Move(in := 65, out1 => "PREMIXING DB"."AUTO BUFF")
   END_RUNG
   RUNG wire#w1
      Contact( "PREMIXING DB".BIT."MATERIAL ADDITION"."MATERIAL SKIP" )
      Move(in := 145, out1 => "PREMIXING DB"."AUTO BUFF")
   END_RUNG
   RUNG wire#powerrail
      { S7_Templates := "SrcType := Int" } NE_Contact(in1 := "PREMIXING DB"."AUTO BUFF", in2 := 60)
      wire#w2
      R_Coil( "PREMIXING DB".BIT."MATERIAL ADDITION"."MATERIAL SELECT" )
   END_RUNG
   RUNG wire#w2
      R_Coil( "PREMIXING DB".BIT."MATERIAL ADDITION"."MATERIAL SKIP" )
   END_RUNG
   // the same network as SCL:
   #_w1 := "AlwaysTRUE" AND NOT "PREMIXING DB".PAUSE AND ("PREMIXING DB"."AUTO BUFF" = 60) AND ("CONTINUE DB"."PREMIXING PROCESS ERROR" <> 1);
   IF #_w1 AND "PREMIXING DB".BIT."MATERIAL ADDITION"."MATERIAL SELECT" THEN
       "PREMIXING DB"."AUTO BUFF" := 65;
   END_IF;
   IF #_w1 AND "PREMIXING DB".BIT."MATERIAL ADDITION"."MATERIAL SKIP" THEN
       "PREMIXING DB"."AUTO BUFF" := 145;
   END_IF;
   IF "PREMIXING DB"."AUTO BUFF" <> 60 THEN
       "PREMIXING DB".BIT."MATERIAL ADDITION"."MATERIAL SELECT" := FALSE;
       "PREMIXING DB".BIT."MATERIAL ADDITION"."MATERIAL SKIP" := FALSE;
   END_IF;
END_REGION

REGION Network 18: ON THE SCREEN FOR MATERIAL ADDITION
   RUNG wire#powerrail
      Contact( "AlwaysTRUE" )
      I_Contact( "PREMIXING DB".PAUSE )
      { S7_Templates := "SrcType := Int" } EQ_Contact(in1 := "PREMIXING DB"."AUTO BUFF", in2 := 65)
      { S7_Templates := "SrcType := Int" } NE_Contact(in1 := "CONTINUE DB"."PREMIXING PROCESS ERROR", in2 := 1)
      Contact( "PREMIXING DB".BIT."MATERIAL ADDITION"."MATERIAL ADDED" )
      Move(in := 70, out1 => "PREMIXING DB"."AUTO BUFF")
   END_RUNG
   RUNG wire#powerrail
      { S7_Templates := "SrcType := Int" } NE_Contact(in1 := "PREMIXING DB"."AUTO BUFF", in2 := 65)
      R_Coil( "PREMIXING DB".BIT."MATERIAL ADDITION"."MATERIAL ADDED" )
   END_RUNG
   // the same network as SCL:
   IF "AlwaysTRUE" AND NOT "PREMIXING DB".PAUSE AND ("PREMIXING DB"."AUTO BUFF" = 65) AND ("CONTINUE DB"."PREMIXING PROCESS ERROR" <> 1) AND "PREMIXING DB".BIT."MATERIAL ADDITION"."MATERIAL ADDED" THEN
       "PREMIXING DB"."AUTO BUFF" := 70;
   END_IF;
   IF "PREMIXING DB"."AUTO BUFF" <> 65 THEN
       "PREMIXING DB".BIT."MATERIAL ADDITION"."MATERIAL ADDED" := FALSE;
   END_IF;
END_REGION

REGION Network 19: ON THE SCREEN FOR MATERIAL ADDITION
   RUNG wire#powerrail
      Contact( "AlwaysTRUE" )
      I_Contact( "PREMIXING DB".PAUSE )
      { S7_Templates := "SrcType := Int" } EQ_Contact(in1 := "PREMIXING DB"."AUTO BUFF", in2 := 70)
      { S7_Templates := "SrcType := Int" } NE_Contact(in1 := "CONTINUE DB"."PREMIXING PROCESS ERROR", in2 := 1)
      { S7_Templates := "time_type := Time" } "IEC_Timer_0_DB_44".TON(pt := T#2S, et =>)
      Move(in := 75, out1 => "PREMIXING DB"."AUTO BUFF")
   END_RUNG
   // the same network as SCL:
   "IEC_Timer_0_DB_44".TON(IN := "AlwaysTRUE" AND NOT "PREMIXING DB".PAUSE AND ("PREMIXING DB"."AUTO BUFF" = 70) AND ("CONTINUE DB"."PREMIXING PROCESS ERROR" <> 1),
                           PT := T#2S);
   IF "IEC_Timer_0_DB_44".Q THEN "PREMIXING DB"."AUTO BUFF" := 75; END_IF;
END_REGION

REGION Network 20: DO YOU WANT TO ADD SORBITOL START / SKIP
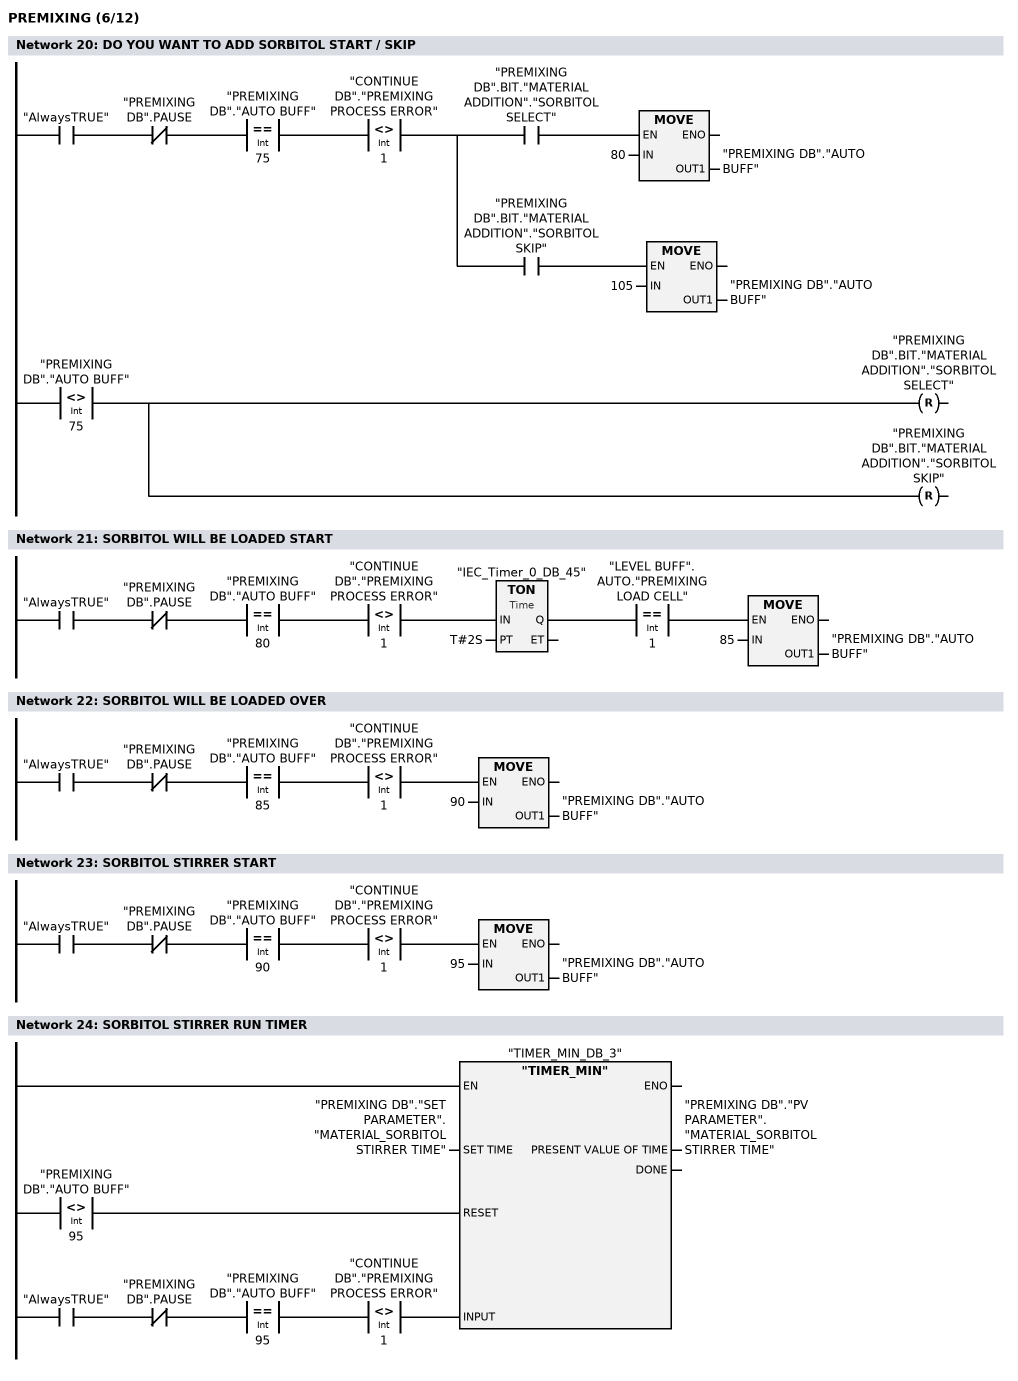
   RUNG wire#powerrail
      Contact( "AlwaysTRUE" )
      I_Contact( "PREMIXING DB".PAUSE )
      { S7_Templates := "SrcType := Int" } EQ_Contact(in1 := "PREMIXING DB"."AUTO BUFF", in2 := 75)
      { S7_Templates := "SrcType := Int" } NE_Contact(in1 := "CONTINUE DB"."PREMIXING PROCESS ERROR", in2 := 1)
      wire#w1
      Contact( "PREMIXING DB".BIT."MATERIAL ADDITION"."SORBITOL SELECT" )
      Move(in := 80, out1 => "PREMIXING DB"."AUTO BUFF")
   END_RUNG
   RUNG wire#w1
      Contact( "PREMIXING DB".BIT."MATERIAL ADDITION"."SORBITOL SKIP" )
      Move(in := 105, out1 => "PREMIXING DB"."AUTO BUFF")
   END_RUNG
   RUNG wire#powerrail
      { S7_Templates := "SrcType := Int" } NE_Contact(in1 := "PREMIXING DB"."AUTO BUFF", in2 := 75)
      wire#w2
      R_Coil( "PREMIXING DB".BIT."MATERIAL ADDITION"."SORBITOL SELECT" )
   END_RUNG
   RUNG wire#w2
      R_Coil( "PREMIXING DB".BIT."MATERIAL ADDITION"."SORBITOL SKIP" )
   END_RUNG
   // the same network as SCL:
   #_w1 := "AlwaysTRUE" AND NOT "PREMIXING DB".PAUSE AND ("PREMIXING DB"."AUTO BUFF" = 75) AND ("CONTINUE DB"."PREMIXING PROCESS ERROR" <> 1);
   IF #_w1 AND "PREMIXING DB".BIT."MATERIAL ADDITION"."SORBITOL SELECT" THEN
       "PREMIXING DB"."AUTO BUFF" := 80;
   END_IF;
   IF #_w1 AND "PREMIXING DB".BIT."MATERIAL ADDITION"."SORBITOL SKIP" THEN
       "PREMIXING DB"."AUTO BUFF" := 105;
   END_IF;
   IF "PREMIXING DB"."AUTO BUFF" <> 75 THEN
       "PREMIXING DB".BIT."MATERIAL ADDITION"."SORBITOL SELECT" := FALSE;
       "PREMIXING DB".BIT."MATERIAL ADDITION"."SORBITOL SKIP" := FALSE;
   END_IF;
END_REGION

REGION Network 21: SORBITOL WILL BE LOADED START
   RUNG wire#powerrail
      Contact( "AlwaysTRUE" )
      I_Contact( "PREMIXING DB".PAUSE )
      { S7_Templates := "SrcType := Int" } EQ_Contact(in1 := "PREMIXING DB"."AUTO BUFF", in2 := 80)
      { S7_Templates := "SrcType := Int" } NE_Contact(in1 := "CONTINUE DB"."PREMIXING PROCESS ERROR", in2 := 1)
      { S7_Templates := "time_type := Time" } "IEC_Timer_0_DB_45".TON(pt := T#2S, et =>)
      { S7_Templates := "SrcType := Int" } EQ_Contact(in1 := "LEVEL BUFF".AUTO."PREMIXING LOAD CELL", in2 := 1)
      Move(in := 85, out1 => "PREMIXING DB"."AUTO BUFF")
   END_RUNG
   // the same network as SCL:
   "IEC_Timer_0_DB_45".TON(IN := "AlwaysTRUE" AND NOT "PREMIXING DB".PAUSE AND ("PREMIXING DB"."AUTO BUFF" = 80) AND ("CONTINUE DB"."PREMIXING PROCESS ERROR" <> 1),
                           PT := T#2S);
   IF "IEC_Timer_0_DB_45".Q AND ("LEVEL BUFF".AUTO."PREMIXING LOAD CELL" = 1) THEN
       "PREMIXING DB"."AUTO BUFF" := 85;
   END_IF;
END_REGION

REGION Network 22: SORBITOL WILL BE LOADED OVER
   RUNG wire#powerrail
      Contact( "AlwaysTRUE" )
      I_Contact( "PREMIXING DB".PAUSE )
      { S7_Templates := "SrcType := Int" } EQ_Contact(in1 := "PREMIXING DB"."AUTO BUFF", in2 := 85)
      { S7_Templates := "SrcType := Int" } NE_Contact(in1 := "CONTINUE DB"."PREMIXING PROCESS ERROR", in2 := 1)
      Move(in := 90, out1 => "PREMIXING DB"."AUTO BUFF")
   END_RUNG
   // the same network as SCL:
   IF "AlwaysTRUE" AND NOT "PREMIXING DB".PAUSE AND ("PREMIXING DB"."AUTO BUFF" = 85) AND ("CONTINUE DB"."PREMIXING PROCESS ERROR" <> 1) THEN
       "PREMIXING DB"."AUTO BUFF" := 90;
   END_IF;
END_REGION

REGION Network 23: SORBITOL STIRRER START
   RUNG wire#powerrail
      Contact( "AlwaysTRUE" )
      I_Contact( "PREMIXING DB".PAUSE )
      { S7_Templates := "SrcType := Int" } EQ_Contact(in1 := "PREMIXING DB"."AUTO BUFF", in2 := 90)
      { S7_Templates := "SrcType := Int" } NE_Contact(in1 := "CONTINUE DB"."PREMIXING PROCESS ERROR", in2 := 1)
      Move(in := 95, out1 => "PREMIXING DB"."AUTO BUFF")
   END_RUNG
   // the same network as SCL:
   IF "AlwaysTRUE" AND NOT "PREMIXING DB".PAUSE AND ("PREMIXING DB"."AUTO BUFF" = 90) AND ("CONTINUE DB"."PREMIXING PROCESS ERROR" <> 1) THEN
       "PREMIXING DB"."AUTO BUFF" := 95;
   END_IF;
END_REGION

REGION Network 24: SORBITOL STIRRER RUN TIMER
   RUNG wire#powerrail
      "TIMER_MIN_DB_3"(RESET := wire#w1, INPUT := wire#w2, "SET TIME" := "PREMIXING DB"."SET PARAMETER"."MATERIAL_SORBITOL STIRRER TIME", "PRESENT VALUE OF TIME" => "PREMIXING DB"."PV PARAMETER"."MATERIAL_SORBITOL STIRRER TIME", DONE =>)
   END_RUNG
   RUNG wire#powerrail
      { S7_Templates := "SrcType := Int" } NE_Contact(in1 := "PREMIXING DB"."AUTO BUFF", in2 := 95)
   END_RUNG wire#w1
   RUNG wire#powerrail
      Contact( "AlwaysTRUE" )
      I_Contact( "PREMIXING DB".PAUSE )
      { S7_Templates := "SrcType := Int" } EQ_Contact(in1 := "PREMIXING DB"."AUTO BUFF", in2 := 95)
      { S7_Templates := "SrcType := Int" } NE_Contact(in1 := "CONTINUE DB"."PREMIXING PROCESS ERROR", in2 := 1)
   END_RUNG wire#w2
   // the same network as SCL:
   "TIMER_MIN_DB_3"("SET TIME" := "PREMIXING DB"."SET PARAMETER"."MATERIAL_SORBITOL STIRRER TIME",   // "TIMER_MIN"
                    RESET := "PREMIXING DB"."AUTO BUFF" <> 95,
                    INPUT := "AlwaysTRUE" AND NOT "PREMIXING DB".PAUSE AND ("PREMIXING DB"."AUTO BUFF" = 95) AND ("CONTINUE DB"."PREMIXING PROCESS ERROR" <> 1),
                    "PRESENT VALUE OF TIME" => "PREMIXING DB"."PV PARAMETER"."MATERIAL_SORBITOL STIRRER TIME");
END_REGION

REGION Network 25: DONE
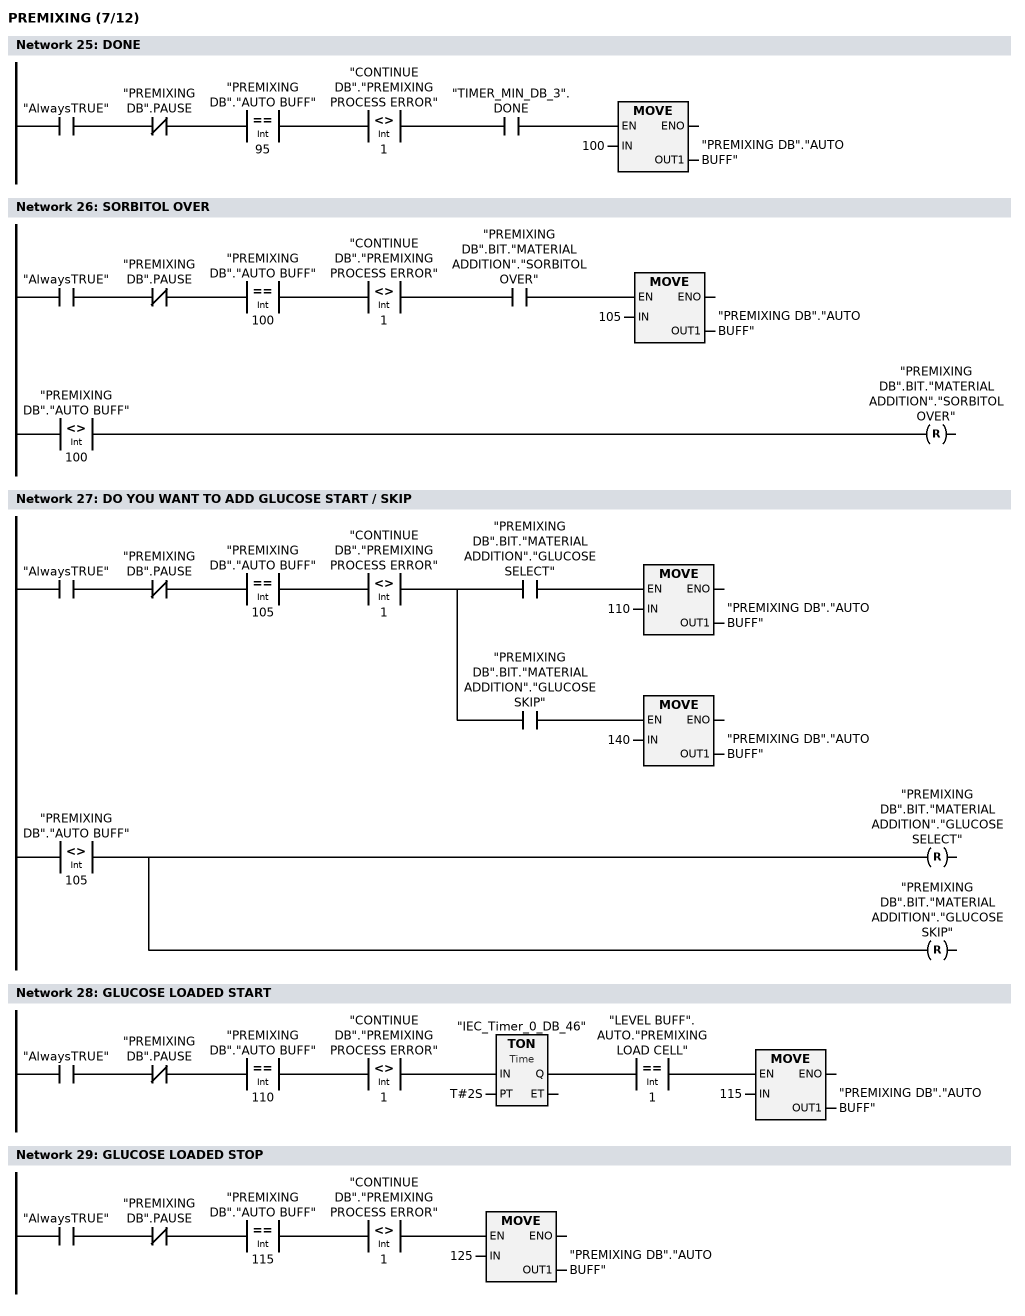
   RUNG wire#powerrail
      Contact( "AlwaysTRUE" )
      I_Contact( "PREMIXING DB".PAUSE )
      { S7_Templates := "SrcType := Int" } EQ_Contact(in1 := "PREMIXING DB"."AUTO BUFF", in2 := 95)
      { S7_Templates := "SrcType := Int" } NE_Contact(in1 := "CONTINUE DB"."PREMIXING PROCESS ERROR", in2 := 1)
      Contact( "TIMER_MIN_DB_3".DONE )
      Move(in := 100, out1 => "PREMIXING DB"."AUTO BUFF")
   END_RUNG
   // the same network as SCL:
   IF "AlwaysTRUE" AND NOT "PREMIXING DB".PAUSE AND ("PREMIXING DB"."AUTO BUFF" = 95) AND ("CONTINUE DB"."PREMIXING PROCESS ERROR" <> 1) AND "TIMER_MIN_DB_3".DONE THEN
       "PREMIXING DB"."AUTO BUFF" := 100;
   END_IF;
END_REGION

REGION Network 26: SORBITOL OVER
   RUNG wire#powerrail
      Contact( "AlwaysTRUE" )
      I_Contact( "PREMIXING DB".PAUSE )
      { S7_Templates := "SrcType := Int" } EQ_Contact(in1 := "PREMIXING DB"."AUTO BUFF", in2 := 100)
      { S7_Templates := "SrcType := Int" } NE_Contact(in1 := "CONTINUE DB"."PREMIXING PROCESS ERROR", in2 := 1)
      Contact( "PREMIXING DB".BIT."MATERIAL ADDITION"."SORBITOL OVER" )
      Move(in := 105, out1 => "PREMIXING DB"."AUTO BUFF")
   END_RUNG
   RUNG wire#powerrail
      { S7_Templates := "SrcType := Int" } NE_Contact(in1 := "PREMIXING DB"."AUTO BUFF", in2 := 100)
      R_Coil( "PREMIXING DB".BIT."MATERIAL ADDITION"."SORBITOL OVER" )
   END_RUNG
   // the same network as SCL:
   IF "AlwaysTRUE" AND NOT "PREMIXING DB".PAUSE AND ("PREMIXING DB"."AUTO BUFF" = 100) AND ("CONTINUE DB"."PREMIXING PROCESS ERROR" <> 1) AND "PREMIXING DB".BIT."MATERIAL ADDITION"."SORBITOL OVER" THEN
       "PREMIXING DB"."AUTO BUFF" := 105;
   END_IF;
   IF "PREMIXING DB"."AUTO BUFF" <> 100 THEN
       "PREMIXING DB".BIT."MATERIAL ADDITION"."SORBITOL OVER" := FALSE;
   END_IF;
END_REGION

REGION Network 27: DO YOU WANT TO ADD GLUCOSE START / SKIP
   RUNG wire#powerrail
      Contact( "AlwaysTRUE" )
      I_Contact( "PREMIXING DB".PAUSE )
      { S7_Templates := "SrcType := Int" } EQ_Contact(in1 := "PREMIXING DB"."AUTO BUFF", in2 := 105)
      { S7_Templates := "SrcType := Int" } NE_Contact(in1 := "CONTINUE DB"."PREMIXING PROCESS ERROR", in2 := 1)
      wire#w1
      Contact( "PREMIXING DB".BIT."MATERIAL ADDITION"."GLUCOSE SELECT" )
      Move(in := 110, out1 => "PREMIXING DB"."AUTO BUFF")
   END_RUNG
   RUNG wire#w1
      Contact( "PREMIXING DB".BIT."MATERIAL ADDITION"."GLUCOSE SKIP" )
      Move(in := 140, out1 => "PREMIXING DB"."AUTO BUFF")
   END_RUNG
   RUNG wire#powerrail
      { S7_Templates := "SrcType := Int" } NE_Contact(in1 := "PREMIXING DB"."AUTO BUFF", in2 := 105)
      wire#w2
      R_Coil( "PREMIXING DB".BIT."MATERIAL ADDITION"."GLUCOSE SELECT" )
   END_RUNG
   RUNG wire#w2
      R_Coil( "PREMIXING DB".BIT."MATERIAL ADDITION"."GLUCOSE SKIP" )
   END_RUNG
   // the same network as SCL:
   #_w1 := "AlwaysTRUE" AND NOT "PREMIXING DB".PAUSE AND ("PREMIXING DB"."AUTO BUFF" = 105) AND ("CONTINUE DB"."PREMIXING PROCESS ERROR" <> 1);
   IF #_w1 AND "PREMIXING DB".BIT."MATERIAL ADDITION"."GLUCOSE SELECT" THEN
       "PREMIXING DB"."AUTO BUFF" := 110;
   END_IF;
   IF #_w1 AND "PREMIXING DB".BIT."MATERIAL ADDITION"."GLUCOSE SKIP" THEN
       "PREMIXING DB"."AUTO BUFF" := 140;
   END_IF;
   IF "PREMIXING DB"."AUTO BUFF" <> 105 THEN
       "PREMIXING DB".BIT."MATERIAL ADDITION"."GLUCOSE SELECT" := FALSE;
       "PREMIXING DB".BIT."MATERIAL ADDITION"."GLUCOSE SKIP" := FALSE;
   END_IF;
END_REGION

REGION Network 28: GLUCOSE LOADED START
   RUNG wire#powerrail
      Contact( "AlwaysTRUE" )
      I_Contact( "PREMIXING DB".PAUSE )
      { S7_Templates := "SrcType := Int" } EQ_Contact(in1 := "PREMIXING DB"."AUTO BUFF", in2 := 110)
      { S7_Templates := "SrcType := Int" } NE_Contact(in1 := "CONTINUE DB"."PREMIXING PROCESS ERROR", in2 := 1)
      { S7_Templates := "time_type := Time" } "IEC_Timer_0_DB_46".TON(pt := T#2S, et =>)
      { S7_Templates := "SrcType := Int" } EQ_Contact(in1 := "LEVEL BUFF".AUTO."PREMIXING LOAD CELL", in2 := 1)
      Move(in := 115, out1 => "PREMIXING DB"."AUTO BUFF")
   END_RUNG
   // the same network as SCL:
   "IEC_Timer_0_DB_46".TON(IN := "AlwaysTRUE" AND NOT "PREMIXING DB".PAUSE AND ("PREMIXING DB"."AUTO BUFF" = 110) AND ("CONTINUE DB"."PREMIXING PROCESS ERROR" <> 1),
                           PT := T#2S);
   IF "IEC_Timer_0_DB_46".Q AND ("LEVEL BUFF".AUTO."PREMIXING LOAD CELL" = 1) THEN
       "PREMIXING DB"."AUTO BUFF" := 115;
   END_IF;
END_REGION

REGION Network 29: GLUCOSE LOADED STOP
   RUNG wire#powerrail
      Contact( "AlwaysTRUE" )
      I_Contact( "PREMIXING DB".PAUSE )
      { S7_Templates := "SrcType := Int" } EQ_Contact(in1 := "PREMIXING DB"."AUTO BUFF", in2 := 115)
      { S7_Templates := "SrcType := Int" } NE_Contact(in1 := "CONTINUE DB"."PREMIXING PROCESS ERROR", in2 := 1)
      Move(in := 125, out1 => "PREMIXING DB"."AUTO BUFF")
   END_RUNG
   // the same network as SCL:
   IF "AlwaysTRUE" AND NOT "PREMIXING DB".PAUSE AND ("PREMIXING DB"."AUTO BUFF" = 115) AND ("CONTINUE DB"."PREMIXING PROCESS ERROR" <> 1) THEN
       "PREMIXING DB"."AUTO BUFF" := 125;
   END_IF;
END_REGION

REGION Network 30: GLUCOSE STIRRER START
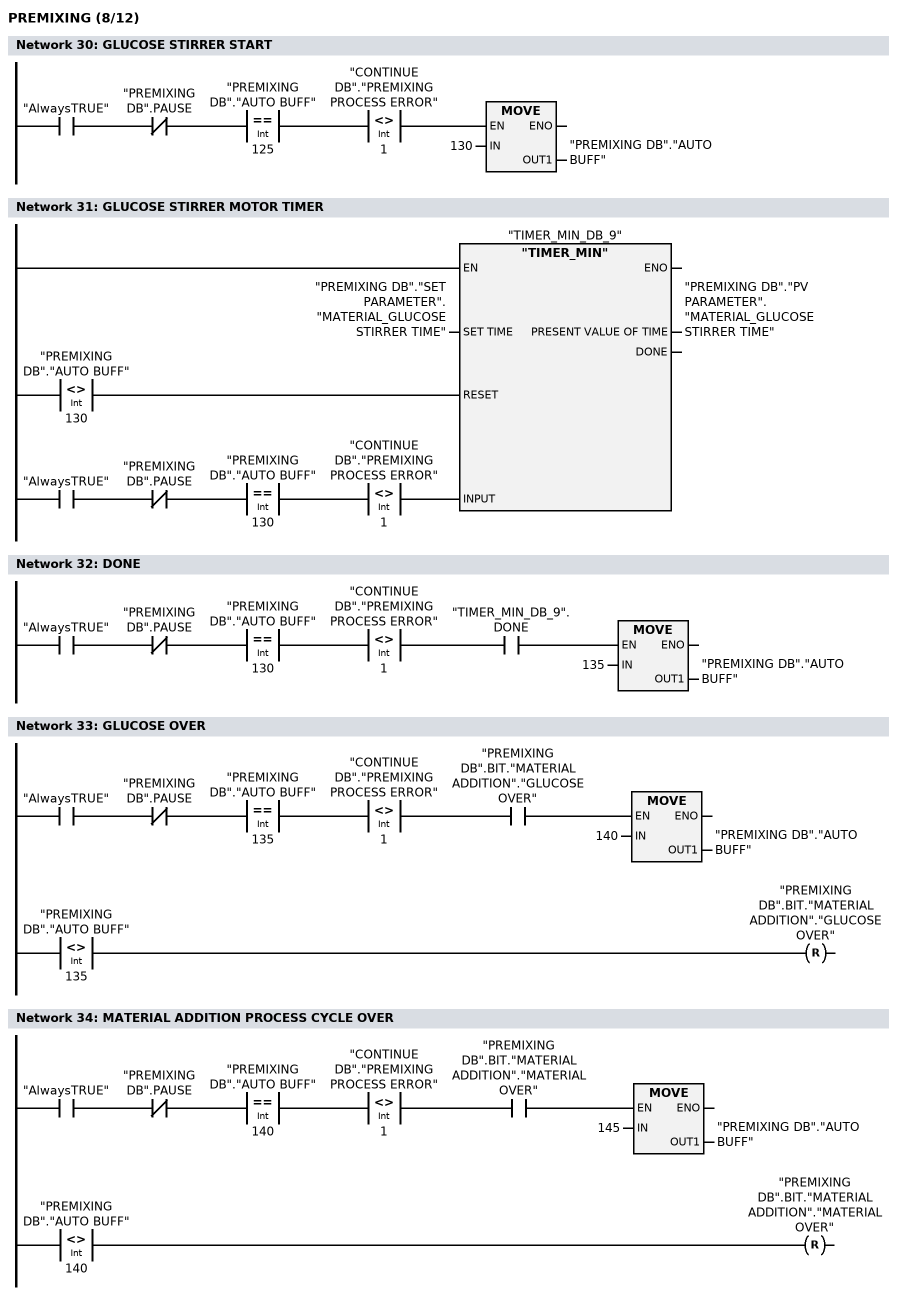
   RUNG wire#powerrail
      Contact( "AlwaysTRUE" )
      I_Contact( "PREMIXING DB".PAUSE )
      { S7_Templates := "SrcType := Int" } EQ_Contact(in1 := "PREMIXING DB"."AUTO BUFF", in2 := 125)
      { S7_Templates := "SrcType := Int" } NE_Contact(in1 := "CONTINUE DB"."PREMIXING PROCESS ERROR", in2 := 1)
      Move(in := 130, out1 => "PREMIXING DB"."AUTO BUFF")
   END_RUNG
   // the same network as SCL:
   IF "AlwaysTRUE" AND NOT "PREMIXING DB".PAUSE AND ("PREMIXING DB"."AUTO BUFF" = 125) AND ("CONTINUE DB"."PREMIXING PROCESS ERROR" <> 1) THEN
       "PREMIXING DB"."AUTO BUFF" := 130;
   END_IF;
END_REGION

REGION Network 31: GLUCOSE STIRRER MOTOR TIMER
   RUNG wire#powerrail
      "TIMER_MIN_DB_9"(RESET := wire#w1, INPUT := wire#w2, "SET TIME" := "PREMIXING DB"."SET PARAMETER"."MATERIAL_GLUCOSE STIRRER TIME", "PRESENT VALUE OF TIME" => "PREMIXING DB"."PV PARAMETER"."MATERIAL_GLUCOSE STIRRER TIME", DONE =>)
   END_RUNG
   RUNG wire#powerrail
      { S7_Templates := "SrcType := Int" } NE_Contact(in1 := "PREMIXING DB"."AUTO BUFF", in2 := 130)
   END_RUNG wire#w1
   RUNG wire#powerrail
      Contact( "AlwaysTRUE" )
      I_Contact( "PREMIXING DB".PAUSE )
      { S7_Templates := "SrcType := Int" } EQ_Contact(in1 := "PREMIXING DB"."AUTO BUFF", in2 := 130)
      { S7_Templates := "SrcType := Int" } NE_Contact(in1 := "CONTINUE DB"."PREMIXING PROCESS ERROR", in2 := 1)
   END_RUNG wire#w2
   // the same network as SCL:
   "TIMER_MIN_DB_9"("SET TIME" := "PREMIXING DB"."SET PARAMETER"."MATERIAL_GLUCOSE STIRRER TIME",   // "TIMER_MIN"
                    RESET := "PREMIXING DB"."AUTO BUFF" <> 130,
                    INPUT := "AlwaysTRUE" AND NOT "PREMIXING DB".PAUSE AND ("PREMIXING DB"."AUTO BUFF" = 130) AND ("CONTINUE DB"."PREMIXING PROCESS ERROR" <> 1),
                    "PRESENT VALUE OF TIME" => "PREMIXING DB"."PV PARAMETER"."MATERIAL_GLUCOSE STIRRER TIME");
END_REGION

REGION Network 32: DONE
   RUNG wire#powerrail
      Contact( "AlwaysTRUE" )
      I_Contact( "PREMIXING DB".PAUSE )
      { S7_Templates := "SrcType := Int" } EQ_Contact(in1 := "PREMIXING DB"."AUTO BUFF", in2 := 130)
      { S7_Templates := "SrcType := Int" } NE_Contact(in1 := "CONTINUE DB"."PREMIXING PROCESS ERROR", in2 := 1)
      Contact( "TIMER_MIN_DB_9".DONE )
      Move(in := 135, out1 => "PREMIXING DB"."AUTO BUFF")
   END_RUNG
   // the same network as SCL:
   IF "AlwaysTRUE" AND NOT "PREMIXING DB".PAUSE AND ("PREMIXING DB"."AUTO BUFF" = 130) AND ("CONTINUE DB"."PREMIXING PROCESS ERROR" <> 1) AND "TIMER_MIN_DB_9".DONE THEN
       "PREMIXING DB"."AUTO BUFF" := 135;
   END_IF;
END_REGION

REGION Network 33: GLUCOSE OVER
   RUNG wire#powerrail
      Contact( "AlwaysTRUE" )
      I_Contact( "PREMIXING DB".PAUSE )
      { S7_Templates := "SrcType := Int" } EQ_Contact(in1 := "PREMIXING DB"."AUTO BUFF", in2 := 135)
      { S7_Templates := "SrcType := Int" } NE_Contact(in1 := "CONTINUE DB"."PREMIXING PROCESS ERROR", in2 := 1)
      Contact( "PREMIXING DB".BIT."MATERIAL ADDITION"."GLUCOSE OVER" )
      Move(in := 140, out1 => "PREMIXING DB"."AUTO BUFF")
   END_RUNG
   RUNG wire#powerrail
      { S7_Templates := "SrcType := Int" } NE_Contact(in1 := "PREMIXING DB"."AUTO BUFF", in2 := 135)
      R_Coil( "PREMIXING DB".BIT."MATERIAL ADDITION"."GLUCOSE OVER" )
   END_RUNG
   // the same network as SCL:
   IF "AlwaysTRUE" AND NOT "PREMIXING DB".PAUSE AND ("PREMIXING DB"."AUTO BUFF" = 135) AND ("CONTINUE DB"."PREMIXING PROCESS ERROR" <> 1) AND "PREMIXING DB".BIT."MATERIAL ADDITION"."GLUCOSE OVER" THEN
       "PREMIXING DB"."AUTO BUFF" := 140;
   END_IF;
   IF "PREMIXING DB"."AUTO BUFF" <> 135 THEN
       "PREMIXING DB".BIT."MATERIAL ADDITION"."GLUCOSE OVER" := FALSE;
   END_IF;
END_REGION

REGION Network 34: MATERIAL ADDITION PROCESS CYCLE OVER
   RUNG wire#powerrail
      Contact( "AlwaysTRUE" )
      I_Contact( "PREMIXING DB".PAUSE )
      { S7_Templates := "SrcType := Int" } EQ_Contact(in1 := "PREMIXING DB"."AUTO BUFF", in2 := 140)
      { S7_Templates := "SrcType := Int" } NE_Contact(in1 := "CONTINUE DB"."PREMIXING PROCESS ERROR", in2 := 1)
      Contact( "PREMIXING DB".BIT."MATERIAL ADDITION"."MATERIAL OVER" )
      Move(in := 145, out1 => "PREMIXING DB"."AUTO BUFF")
   END_RUNG
   RUNG wire#powerrail
      { S7_Templates := "SrcType := Int" } NE_Contact(in1 := "PREMIXING DB"."AUTO BUFF", in2 := 140)
      R_Coil( "PREMIXING DB".BIT."MATERIAL ADDITION"."MATERIAL OVER" )
   END_RUNG
   // the same network as SCL:
   IF "AlwaysTRUE" AND NOT "PREMIXING DB".PAUSE AND ("PREMIXING DB"."AUTO BUFF" = 140) AND ("CONTINUE DB"."PREMIXING PROCESS ERROR" <> 1) AND "PREMIXING DB".BIT."MATERIAL ADDITION"."MATERIAL OVER" THEN
       "PREMIXING DB"."AUTO BUFF" := 145;
   END_IF;
   IF "PREMIXING DB"."AUTO BUFF" <> 140 THEN
       "PREMIXING DB".BIT."MATERIAL ADDITION"."MATERIAL OVER" := FALSE;
   END_IF;
END_REGION

REGION Network 36: RECIRCULATION SELECT
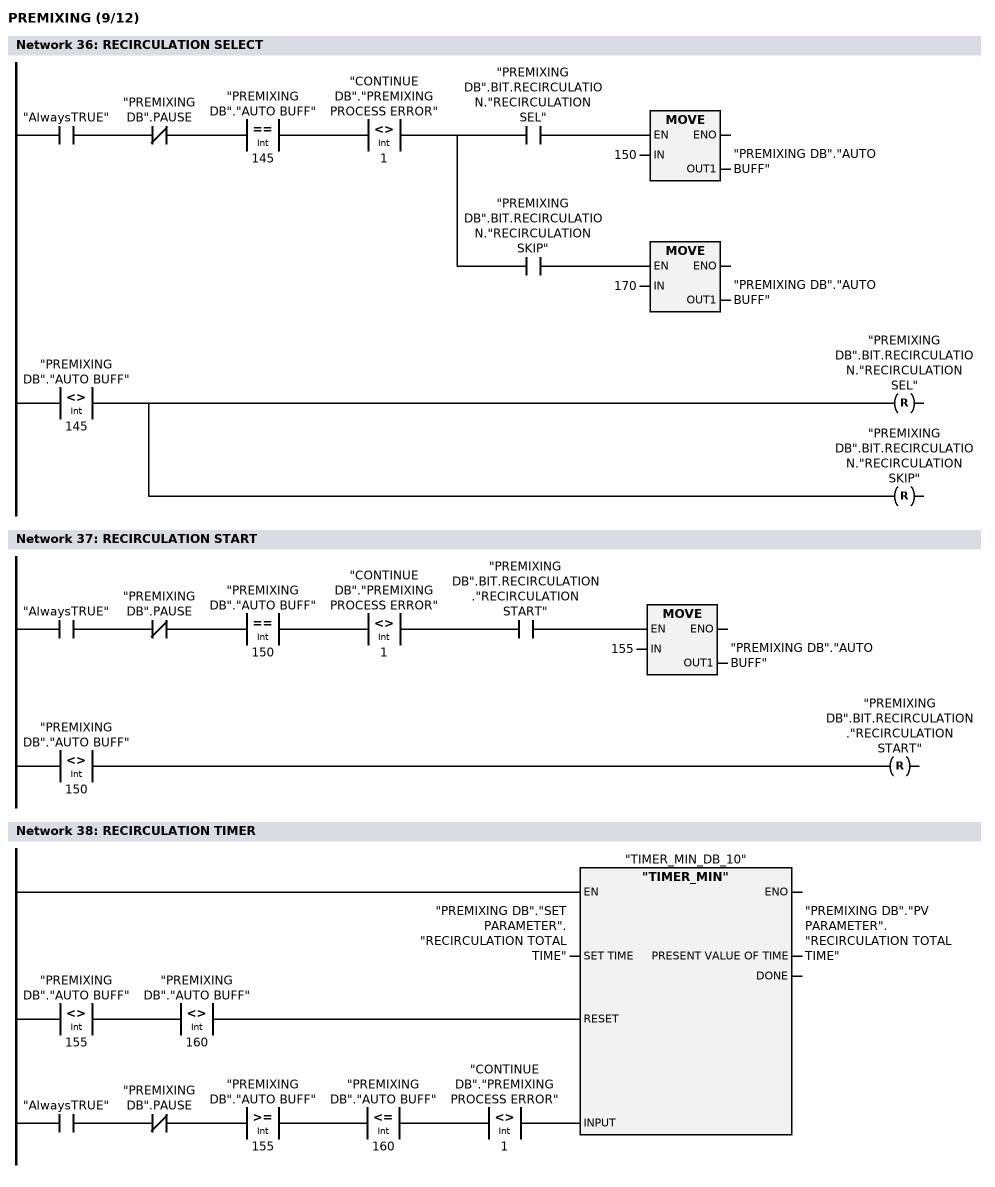
   RUNG wire#powerrail
      Contact( "AlwaysTRUE" )
      I_Contact( "PREMIXING DB".PAUSE )
      { S7_Templates := "SrcType := Int" } EQ_Contact(in1 := "PREMIXING DB"."AUTO BUFF", in2 := 145)
      { S7_Templates := "SrcType := Int" } NE_Contact(in1 := "CONTINUE DB"."PREMIXING PROCESS ERROR", in2 := 1)
      wire#w1
      Contact( "PREMIXING DB".BIT.RECIRCULATION."RECIRCULATION SEL" )
      Move(in := 150, out1 => "PREMIXING DB"."AUTO BUFF")
   END_RUNG
   RUNG wire#w1
      Contact( "PREMIXING DB".BIT.RECIRCULATION."RECIRCULATION SKIP" )
      Move(in := 170, out1 => "PREMIXING DB"."AUTO BUFF")
   END_RUNG
   RUNG wire#powerrail
      { S7_Templates := "SrcType := Int" } NE_Contact(in1 := "PREMIXING DB"."AUTO BUFF", in2 := 145)
      wire#w2
      R_Coil( "PREMIXING DB".BIT.RECIRCULATION."RECIRCULATION SEL" )
   END_RUNG
   RUNG wire#w2
      R_Coil( "PREMIXING DB".BIT.RECIRCULATION."RECIRCULATION SKIP" )
   END_RUNG
   // the same network as SCL:
   #_w1 := "AlwaysTRUE" AND NOT "PREMIXING DB".PAUSE AND ("PREMIXING DB"."AUTO BUFF" = 145) AND ("CONTINUE DB"."PREMIXING PROCESS ERROR" <> 1);
   IF #_w1 AND "PREMIXING DB".BIT.RECIRCULATION."RECIRCULATION SEL" THEN
       "PREMIXING DB"."AUTO BUFF" := 150;
   END_IF;
   IF #_w1 AND "PREMIXING DB".BIT.RECIRCULATION."RECIRCULATION SKIP" THEN
       "PREMIXING DB"."AUTO BUFF" := 170;
   END_IF;
   IF "PREMIXING DB"."AUTO BUFF" <> 145 THEN
       "PREMIXING DB".BIT.RECIRCULATION."RECIRCULATION SEL" := FALSE;
       "PREMIXING DB".BIT.RECIRCULATION."RECIRCULATION SKIP" := FALSE;
   END_IF;
END_REGION

REGION Network 37: RECIRCULATION START
   RUNG wire#powerrail
      Contact( "AlwaysTRUE" )
      I_Contact( "PREMIXING DB".PAUSE )
      { S7_Templates := "SrcType := Int" } EQ_Contact(in1 := "PREMIXING DB"."AUTO BUFF", in2 := 150)
      { S7_Templates := "SrcType := Int" } NE_Contact(in1 := "CONTINUE DB"."PREMIXING PROCESS ERROR", in2 := 1)
      Contact( "PREMIXING DB".BIT.RECIRCULATION."RECIRCULATION START" )
      Move(in := 155, out1 => "PREMIXING DB"."AUTO BUFF")
   END_RUNG
   RUNG wire#powerrail
      { S7_Templates := "SrcType := Int" } NE_Contact(in1 := "PREMIXING DB"."AUTO BUFF", in2 := 150)
      R_Coil( "PREMIXING DB".BIT.RECIRCULATION."RECIRCULATION START" )
   END_RUNG
   // the same network as SCL:
   IF "AlwaysTRUE" AND NOT "PREMIXING DB".PAUSE AND ("PREMIXING DB"."AUTO BUFF" = 150) AND ("CONTINUE DB"."PREMIXING PROCESS ERROR" <> 1) AND "PREMIXING DB".BIT.RECIRCULATION."RECIRCULATION START" THEN
       "PREMIXING DB"."AUTO BUFF" := 155;
   END_IF;
   IF "PREMIXING DB"."AUTO BUFF" <> 150 THEN
       "PREMIXING DB".BIT.RECIRCULATION."RECIRCULATION START" := FALSE;
   END_IF;
END_REGION

REGION Network 38: RECIRCULATION TIMER
   RUNG wire#powerrail
      "TIMER_MIN_DB_10"(RESET := wire#w1, INPUT := wire#w2, "SET TIME" := "PREMIXING DB"."SET PARAMETER"."RECIRCULATION TOTAL TIME", "PRESENT VALUE OF TIME" => "PREMIXING DB"."PV PARAMETER"."RECIRCULATION TOTAL TIME", DONE =>)
   END_RUNG
   RUNG wire#powerrail
      { S7_Templates := "SrcType := Int" } NE_Contact(in1 := "PREMIXING DB"."AUTO BUFF", in2 := 155)
      { S7_Templates := "SrcType := Int" } NE_Contact(in1 := "PREMIXING DB"."AUTO BUFF", in2 := 160)
   END_RUNG wire#w1
   RUNG wire#powerrail
      Contact( "AlwaysTRUE" )
      I_Contact( "PREMIXING DB".PAUSE )
      { S7_Templates := "SrcType := Int" } GE_Contact(in1 := "PREMIXING DB"."AUTO BUFF", in2 := 155)
      { S7_Templates := "SrcType := Int" } LE_Contact(in1 := "PREMIXING DB"."AUTO BUFF", in2 := 160)
      { S7_Templates := "SrcType := Int" } NE_Contact(in1 := "CONTINUE DB"."PREMIXING PROCESS ERROR", in2 := 1)
   END_RUNG wire#w2
   // the same network as SCL:
   "TIMER_MIN_DB_10"("SET TIME" := "PREMIXING DB"."SET PARAMETER"."RECIRCULATION TOTAL TIME",   // "TIMER_MIN"
                     RESET := ("PREMIXING DB"."AUTO BUFF" <> 155) AND ("PREMIXING DB"."AUTO BUFF" <> 160),
                     INPUT := "AlwaysTRUE" AND NOT "PREMIXING DB".PAUSE AND ("PREMIXING DB"."AUTO BUFF" >= 155) AND ("PREMIXING DB"."AUTO BUFF" <= 160) AND ("CONTINUE DB"."PREMIXING PROCESS ERROR" <> 1),
                     "PRESENT VALUE OF TIME" => "PREMIXING DB"."PV PARAMETER"."RECIRCULATION TOTAL TIME");
END_REGION

REGION Network 39: HOMOGENIZER DELAY TIMER
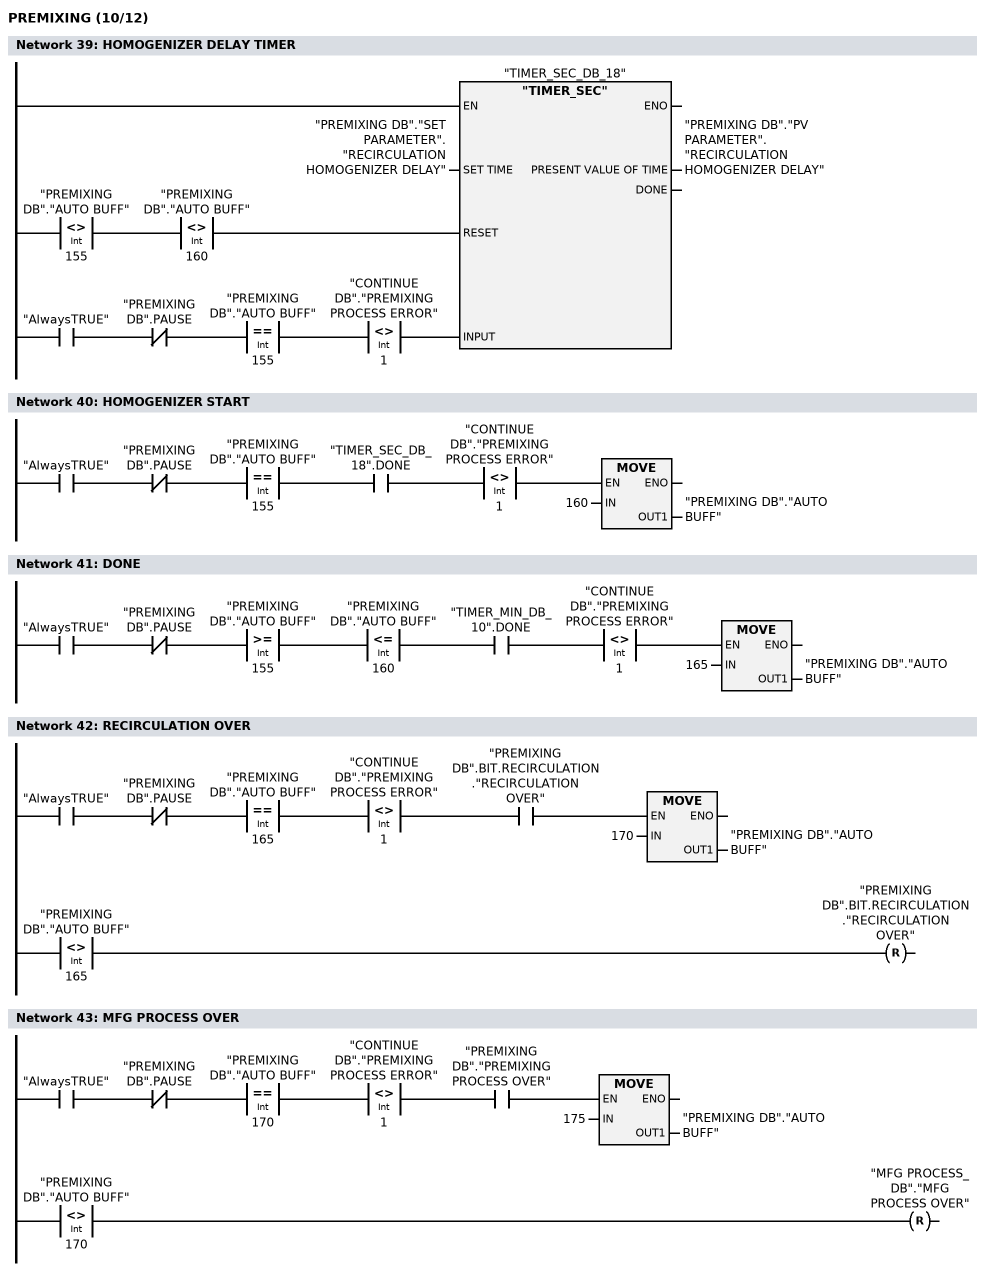
   RUNG wire#powerrail
      "TIMER_SEC_DB_18"(RESET := wire#w1, INPUT := wire#w2, "SET TIME" := "PREMIXING DB"."SET PARAMETER"."RECIRCULATION HOMOGENIZER DELAY", "PRESENT VALUE OF TIME" => "PREMIXING DB"."PV PARAMETER"."RECIRCULATION HOMOGENIZER DELAY", DONE =>)
   END_RUNG
   RUNG wire#powerrail
      { S7_Templates := "SrcType := Int" } NE_Contact(in1 := "PREMIXING DB"."AUTO BUFF", in2 := 155)
      { S7_Templates := "SrcType := Int" } NE_Contact(in1 := "PREMIXING DB"."AUTO BUFF", in2 := 160)
   END_RUNG wire#w1
   RUNG wire#powerrail
      Contact( "AlwaysTRUE" )
      I_Contact( "PREMIXING DB".PAUSE )
      { S7_Templates := "SrcType := Int" } EQ_Contact(in1 := "PREMIXING DB"."AUTO BUFF", in2 := 155)
      { S7_Templates := "SrcType := Int" } NE_Contact(in1 := "CONTINUE DB"."PREMIXING PROCESS ERROR", in2 := 1)
   END_RUNG wire#w2
   // the same network as SCL:
   "TIMER_SEC_DB_18"("SET TIME" := "PREMIXING DB"."SET PARAMETER"."RECIRCULATION HOMOGENIZER DELAY",   // "TIMER_SEC"
                     RESET := ("PREMIXING DB"."AUTO BUFF" <> 155) AND ("PREMIXING DB"."AUTO BUFF" <> 160),
                     INPUT := "AlwaysTRUE" AND NOT "PREMIXING DB".PAUSE AND ("PREMIXING DB"."AUTO BUFF" = 155) AND ("CONTINUE DB"."PREMIXING PROCESS ERROR" <> 1),
                     "PRESENT VALUE OF TIME" => "PREMIXING DB"."PV PARAMETER"."RECIRCULATION HOMOGENIZER DELAY");
END_REGION

REGION Network 40: HOMOGENIZER START
   RUNG wire#powerrail
      Contact( "AlwaysTRUE" )
      I_Contact( "PREMIXING DB".PAUSE )
      { S7_Templates := "SrcType := Int" } EQ_Contact(in1 := "PREMIXING DB"."AUTO BUFF", in2 := 155)
      Contact( "TIMER_SEC_DB_18".DONE )
      { S7_Templates := "SrcType := Int" } NE_Contact(in1 := "CONTINUE DB"."PREMIXING PROCESS ERROR", in2 := 1)
      Move(in := 160, out1 => "PREMIXING DB"."AUTO BUFF")
   END_RUNG
   // the same network as SCL:
   IF "AlwaysTRUE" AND NOT "PREMIXING DB".PAUSE AND ("PREMIXING DB"."AUTO BUFF" = 155) AND "TIMER_SEC_DB_18".DONE AND ("CONTINUE DB"."PREMIXING PROCESS ERROR" <> 1) THEN
       "PREMIXING DB"."AUTO BUFF" := 160;
   END_IF;
END_REGION

REGION Network 41: DONE
   RUNG wire#powerrail
      Contact( "AlwaysTRUE" )
      I_Contact( "PREMIXING DB".PAUSE )
      { S7_Templates := "SrcType := Int" } GE_Contact(in1 := "PREMIXING DB"."AUTO BUFF", in2 := 155)
      { S7_Templates := "SrcType := Int" } LE_Contact(in1 := "PREMIXING DB"."AUTO BUFF", in2 := 160)
      Contact( "TIMER_MIN_DB_10".DONE )
      { S7_Templates := "SrcType := Int" } NE_Contact(in1 := "CONTINUE DB"."PREMIXING PROCESS ERROR", in2 := 1)
      Move(in := 165, out1 => "PREMIXING DB"."AUTO BUFF")
   END_RUNG
   // the same network as SCL:
   IF "AlwaysTRUE" AND NOT "PREMIXING DB".PAUSE AND ("PREMIXING DB"."AUTO BUFF" >= 155) AND ("PREMIXING DB"."AUTO BUFF" <= 160) AND "TIMER_MIN_DB_10".DONE AND ("CONTINUE DB"."PREMIXING PROCESS ERROR" <> 1) THEN
       "PREMIXING DB"."AUTO BUFF" := 165;
   END_IF;
END_REGION

REGION Network 42: RECIRCULATION OVER
   RUNG wire#powerrail
      Contact( "AlwaysTRUE" )
      I_Contact( "PREMIXING DB".PAUSE )
      { S7_Templates := "SrcType := Int" } EQ_Contact(in1 := "PREMIXING DB"."AUTO BUFF", in2 := 165)
      { S7_Templates := "SrcType := Int" } NE_Contact(in1 := "CONTINUE DB"."PREMIXING PROCESS ERROR", in2 := 1)
      Contact( "PREMIXING DB".BIT.RECIRCULATION."RECIRCULATION OVER" )
      Move(in := 170, out1 => "PREMIXING DB"."AUTO BUFF")
   END_RUNG
   RUNG wire#powerrail
      { S7_Templates := "SrcType := Int" } NE_Contact(in1 := "PREMIXING DB"."AUTO BUFF", in2 := 165)
      R_Coil( "PREMIXING DB".BIT.RECIRCULATION."RECIRCULATION OVER" )
   END_RUNG
   // the same network as SCL:
   IF "AlwaysTRUE" AND NOT "PREMIXING DB".PAUSE AND ("PREMIXING DB"."AUTO BUFF" = 165) AND ("CONTINUE DB"."PREMIXING PROCESS ERROR" <> 1) AND "PREMIXING DB".BIT.RECIRCULATION."RECIRCULATION OVER" THEN
       "PREMIXING DB"."AUTO BUFF" := 170;
   END_IF;
   IF "PREMIXING DB"."AUTO BUFF" <> 165 THEN
       "PREMIXING DB".BIT.RECIRCULATION."RECIRCULATION OVER" := FALSE;
   END_IF;
END_REGION

REGION Network 43: MFG PROCESS OVER
   RUNG wire#powerrail
      Contact( "AlwaysTRUE" )
      I_Contact( "PREMIXING DB".PAUSE )
      { S7_Templates := "SrcType := Int" } EQ_Contact(in1 := "PREMIXING DB"."AUTO BUFF", in2 := 170)
      { S7_Templates := "SrcType := Int" } NE_Contact(in1 := "CONTINUE DB"."PREMIXING PROCESS ERROR", in2 := 1)
      Contact( "PREMIXING DB"."PREMIXING PROCESS OVER" )
      Move(in := 175, out1 => "PREMIXING DB"."AUTO BUFF")
   END_RUNG
   RUNG wire#powerrail
      { S7_Templates := "SrcType := Int" } NE_Contact(in1 := "PREMIXING DB"."AUTO BUFF", in2 := 170)
      R_Coil( "MFG PROCESS_DB"."MFG PROCESS OVER" )
   END_RUNG
   // the same network as SCL:
   IF "AlwaysTRUE" AND NOT "PREMIXING DB".PAUSE AND ("PREMIXING DB"."AUTO BUFF" = 170) AND ("CONTINUE DB"."PREMIXING PROCESS ERROR" <> 1) AND "PREMIXING DB"."PREMIXING PROCESS OVER" THEN
       "PREMIXING DB"."AUTO BUFF" := 175;
   END_IF;
   IF "PREMIXING DB"."AUTO BUFF" <> 170 THEN "MFG PROCESS_DB"."MFG PROCESS OVER" := FALSE; END_IF;
END_REGION

REGION Network 44: STOP
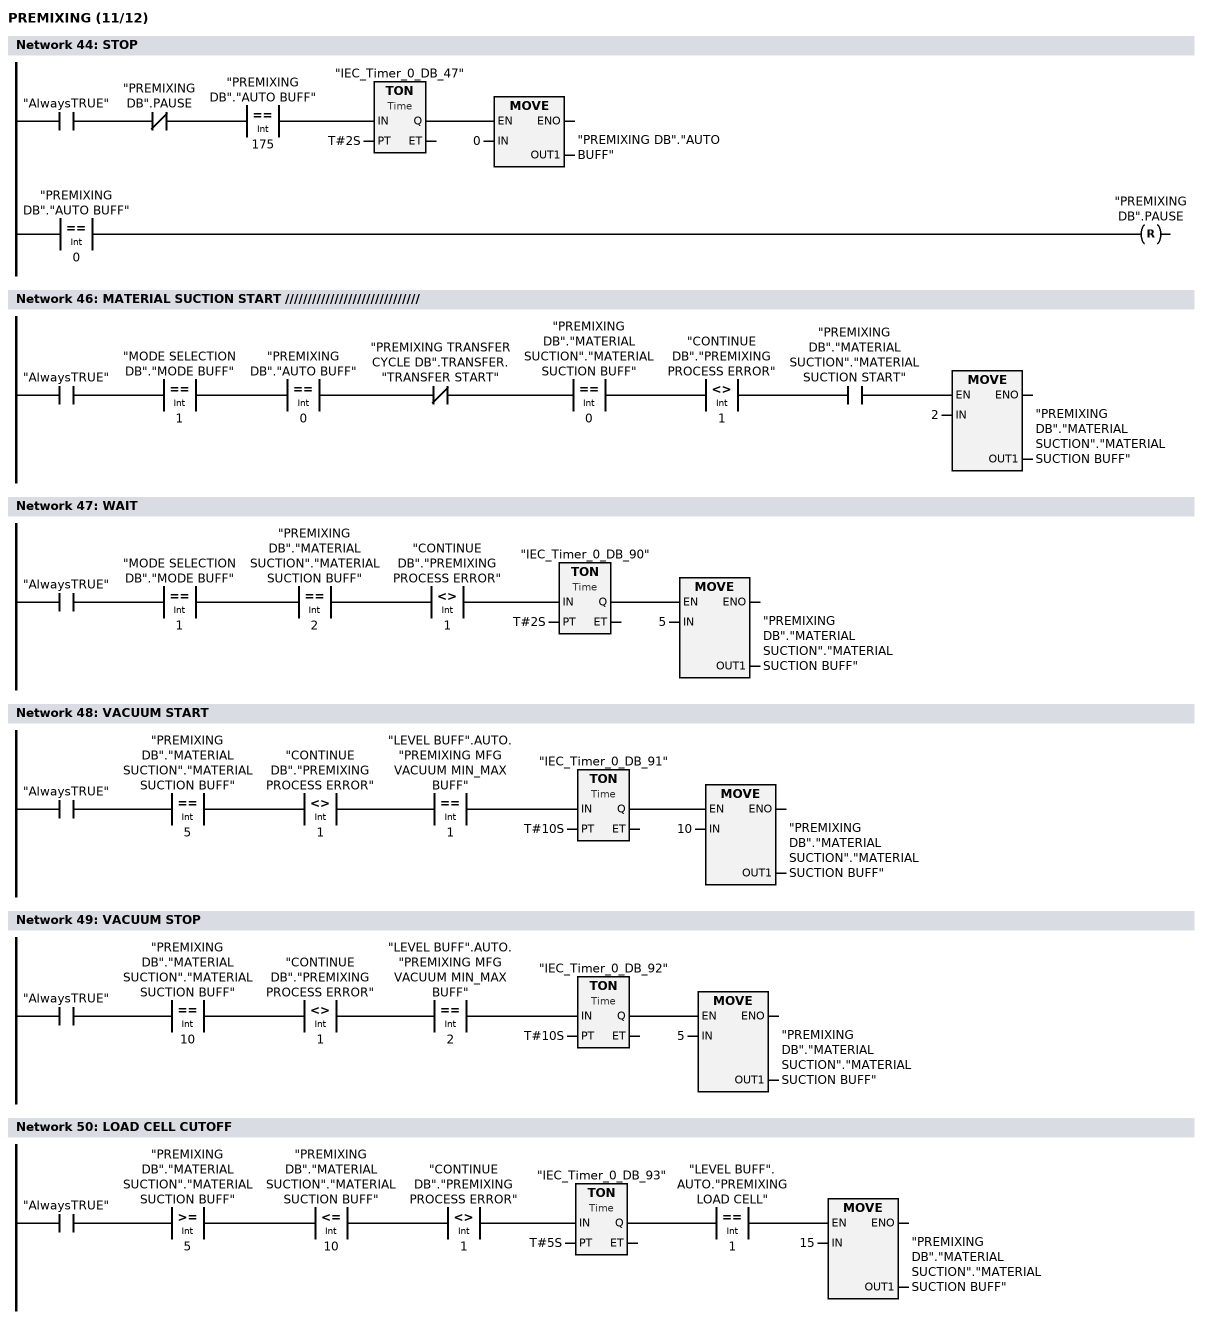
   RUNG wire#powerrail
      Contact( "AlwaysTRUE" )
      I_Contact( "PREMIXING DB".PAUSE )
      { S7_Templates := "SrcType := Int" } EQ_Contact(in1 := "PREMIXING DB"."AUTO BUFF", in2 := 175)
      { S7_Templates := "time_type := Time" } "IEC_Timer_0_DB_47".TON(pt := T#2S, et =>)
      Move(in := 0, out1 => "PREMIXING DB"."AUTO BUFF")
   END_RUNG
   RUNG wire#powerrail
      { S7_Templates := "SrcType := Int" } EQ_Contact(in1 := "PREMIXING DB"."AUTO BUFF", in2 := 0)
      R_Coil( "PREMIXING DB".PAUSE )
   END_RUNG
   // the same network as SCL:
   "IEC_Timer_0_DB_47".TON(IN := "AlwaysTRUE" AND NOT "PREMIXING DB".PAUSE AND ("PREMIXING DB"."AUTO BUFF" = 175),
                           PT := T#2S);
   IF "IEC_Timer_0_DB_47".Q THEN "PREMIXING DB"."AUTO BUFF" := 0; END_IF;
   IF "PREMIXING DB"."AUTO BUFF" = 0 THEN "PREMIXING DB".PAUSE := FALSE; END_IF;
END_REGION

REGION Network 46: MATERIAL SUCTION START //////////////////////////////
   RUNG wire#powerrail
      Contact( "AlwaysTRUE" )
      { S7_Templates := "SrcType := Int" } EQ_Contact(in1 := "MODE SELECTION DB"."MODE BUFF", in2 := 1)
      { S7_Templates := "SrcType := Int" } EQ_Contact(in1 := "PREMIXING DB"."AUTO BUFF", in2 := 0)
      I_Contact( "PREMIXING TRANSFER CYCLE DB".TRANSFER."TRANSFER START" )
      { S7_Templates := "SrcType := Int" } EQ_Contact(in1 := "PREMIXING DB"."MATERIAL SUCTION"."MATERIAL SUCTION BUFF", in2 := 0)
      { S7_Templates := "SrcType := Int" } NE_Contact(in1 := "CONTINUE DB"."PREMIXING PROCESS ERROR", in2 := 1)
      Contact( "PREMIXING DB"."MATERIAL SUCTION"."MATERIAL SUCTION START" )
      Move(in := 2, out1 => "PREMIXING DB"."MATERIAL SUCTION"."MATERIAL SUCTION BUFF")
   END_RUNG
   // the same network as SCL:
   IF "AlwaysTRUE" AND ("MODE SELECTION DB"."MODE BUFF" = 1) AND ("PREMIXING DB"."AUTO BUFF" = 0) AND NOT "PREMIXING TRANSFER CYCLE DB".TRANSFER."TRANSFER START" AND ("PREMIXING DB"."MATERIAL SUCTION"."MATERIAL SUCTION BUFF" = 0) AND ("CONTINUE DB"."PREMIXING PROCESS ERROR" <> 1) AND "PREMIXING DB"."MATERIAL SUCTION"."MATERIAL SUCTION START" THEN
       "PREMIXING DB"."MATERIAL SUCTION"."MATERIAL SUCTION BUFF" := 2;
   END_IF;
END_REGION

REGION Network 47: WAIT
   RUNG wire#powerrail
      Contact( "AlwaysTRUE" )
      { S7_Templates := "SrcType := Int" } EQ_Contact(in1 := "MODE SELECTION DB"."MODE BUFF", in2 := 1)
      { S7_Templates := "SrcType := Int" } EQ_Contact(in1 := "PREMIXING DB"."MATERIAL SUCTION"."MATERIAL SUCTION BUFF", in2 := 2)
      { S7_Templates := "SrcType := Int" } NE_Contact(in1 := "CONTINUE DB"."PREMIXING PROCESS ERROR", in2 := 1)
      { S7_Templates := "time_type := Time" } "IEC_Timer_0_DB_90".TON(pt := T#2S, et =>)
      Move(in := 5, out1 => "PREMIXING DB"."MATERIAL SUCTION"."MATERIAL SUCTION BUFF")
   END_RUNG
   // the same network as SCL:
   "IEC_Timer_0_DB_90".TON(IN := "AlwaysTRUE" AND ("MODE SELECTION DB"."MODE BUFF" = 1) AND ("PREMIXING DB"."MATERIAL SUCTION"."MATERIAL SUCTION BUFF" = 2) AND ("CONTINUE DB"."PREMIXING PROCESS ERROR" <> 1),
                           PT := T#2S);
   IF "IEC_Timer_0_DB_90".Q THEN "PREMIXING DB"."MATERIAL SUCTION"."MATERIAL SUCTION BUFF" := 5; END_IF;
END_REGION

REGION Network 48: VACUUM START
   RUNG wire#powerrail
      Contact( "AlwaysTRUE" )
      { S7_Templates := "SrcType := Int" } EQ_Contact(in1 := "PREMIXING DB"."MATERIAL SUCTION"."MATERIAL SUCTION BUFF", in2 := 5)
      { S7_Templates := "SrcType := Int" } NE_Contact(in1 := "CONTINUE DB"."PREMIXING PROCESS ERROR", in2 := 1)
      { S7_Templates := "SrcType := Int" } EQ_Contact(in1 := "LEVEL BUFF".AUTO."PREMIXING MFG VACUUM MIN_MAX BUFF", in2 := 1)
      { S7_Templates := "time_type := Time" } "IEC_Timer_0_DB_91".TON(pt := T#10S, et =>)
      Move(in := 10, out1 => "PREMIXING DB"."MATERIAL SUCTION"."MATERIAL SUCTION BUFF")
   END_RUNG
   // the same network as SCL:
   "IEC_Timer_0_DB_91".TON(IN := "AlwaysTRUE" AND ("PREMIXING DB"."MATERIAL SUCTION"."MATERIAL SUCTION BUFF" = 5) AND ("CONTINUE DB"."PREMIXING PROCESS ERROR" <> 1) AND ("LEVEL BUFF".AUTO."PREMIXING MFG VACUUM MIN_MAX BUFF" = 1),
                           PT := T#10S);
   IF "IEC_Timer_0_DB_91".Q THEN "PREMIXING DB"."MATERIAL SUCTION"."MATERIAL SUCTION BUFF" := 10; END_IF;
END_REGION

REGION Network 49: VACUUM STOP
   RUNG wire#powerrail
      Contact( "AlwaysTRUE" )
      { S7_Templates := "SrcType := Int" } EQ_Contact(in1 := "PREMIXING DB"."MATERIAL SUCTION"."MATERIAL SUCTION BUFF", in2 := 10)
      { S7_Templates := "SrcType := Int" } NE_Contact(in1 := "CONTINUE DB"."PREMIXING PROCESS ERROR", in2 := 1)
      { S7_Templates := "SrcType := Int" } EQ_Contact(in1 := "LEVEL BUFF".AUTO."PREMIXING MFG VACUUM MIN_MAX BUFF", in2 := 2)
      { S7_Templates := "time_type := Time" } "IEC_Timer_0_DB_92".TON(pt := T#10S, et =>)
      Move(in := 5, out1 => "PREMIXING DB"."MATERIAL SUCTION"."MATERIAL SUCTION BUFF")
   END_RUNG
   // the same network as SCL:
   "IEC_Timer_0_DB_92".TON(IN := "AlwaysTRUE" AND ("PREMIXING DB"."MATERIAL SUCTION"."MATERIAL SUCTION BUFF" = 10) AND ("CONTINUE DB"."PREMIXING PROCESS ERROR" <> 1) AND ("LEVEL BUFF".AUTO."PREMIXING MFG VACUUM MIN_MAX BUFF" = 2),
                           PT := T#10S);
   IF "IEC_Timer_0_DB_92".Q THEN "PREMIXING DB"."MATERIAL SUCTION"."MATERIAL SUCTION BUFF" := 5; END_IF;
END_REGION

REGION Network 50: LOAD CELL CUTOFF
   RUNG wire#powerrail
      Contact( "AlwaysTRUE" )
      { S7_Templates := "SrcType := Int" } GE_Contact(in1 := "PREMIXING DB"."MATERIAL SUCTION"."MATERIAL SUCTION BUFF", in2 := 5)
      { S7_Templates := "SrcType := Int" } LE_Contact(in1 := "PREMIXING DB"."MATERIAL SUCTION"."MATERIAL SUCTION BUFF", in2 := 10)
      { S7_Templates := "SrcType := Int" } NE_Contact(in1 := "CONTINUE DB"."PREMIXING PROCESS ERROR", in2 := 1)
      { S7_Templates := "time_type := Time" } "IEC_Timer_0_DB_93".TON(pt := T#5S, et =>)
      { S7_Templates := "SrcType := Int" } EQ_Contact(in1 := "LEVEL BUFF".AUTO."PREMIXING LOAD CELL", in2 := 1)
      Move(in := 15, out1 => "PREMIXING DB"."MATERIAL SUCTION"."MATERIAL SUCTION BUFF")
   END_RUNG
   // the same network as SCL:
   "IEC_Timer_0_DB_93".TON(IN := "AlwaysTRUE" AND ("PREMIXING DB"."MATERIAL SUCTION"."MATERIAL SUCTION BUFF" >= 5) AND ("PREMIXING DB"."MATERIAL SUCTION"."MATERIAL SUCTION BUFF" <= 10) AND ("CONTINUE DB"."PREMIXING PROCESS ERROR" <> 1),
                           PT := T#5S);
   IF "IEC_Timer_0_DB_93".Q AND ("LEVEL BUFF".AUTO."PREMIXING LOAD CELL" = 1) THEN
       "PREMIXING DB"."MATERIAL SUCTION"."MATERIAL SUCTION BUFF" := 15;
   END_IF;
END_REGION

REGION Network 51: MATERIAL SUCTION OVER
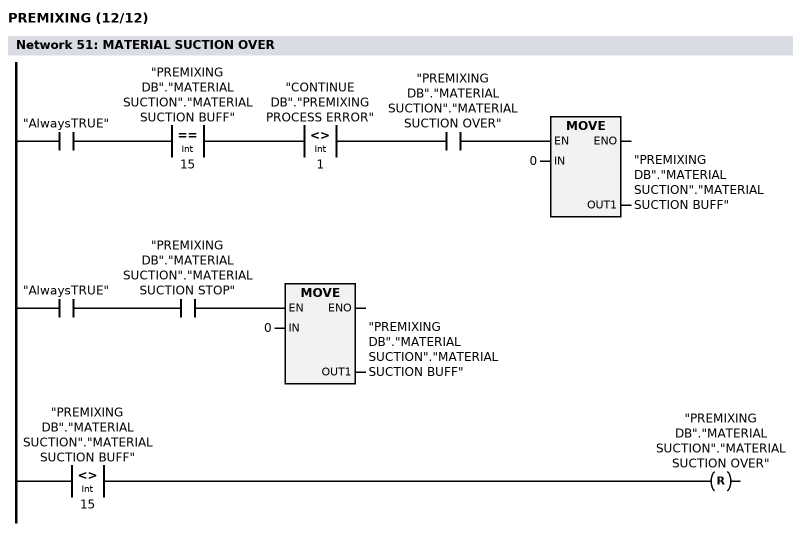
   RUNG wire#powerrail
      Contact( "AlwaysTRUE" )
      { S7_Templates := "SrcType := Int" } EQ_Contact(in1 := "PREMIXING DB"."MATERIAL SUCTION"."MATERIAL SUCTION BUFF", in2 := 15)
      { S7_Templates := "SrcType := Int" } NE_Contact(in1 := "CONTINUE DB"."PREMIXING PROCESS ERROR", in2 := 1)
      Contact( "PREMIXING DB"."MATERIAL SUCTION"."MATERIAL SUCTION OVER" )
      Move(in := 0, out1 => "PREMIXING DB"."MATERIAL SUCTION"."MATERIAL SUCTION BUFF")
   END_RUNG
   RUNG wire#powerrail
      Contact( "AlwaysTRUE" )
      Contact( "PREMIXING DB"."MATERIAL SUCTION"."MATERIAL SUCTION STOP" )
      Move(in := 0, out1 => "PREMIXING DB"."MATERIAL SUCTION"."MATERIAL SUCTION BUFF")
   END_RUNG
   RUNG wire#powerrail
      { S7_Templates := "SrcType := Int" } NE_Contact(in1 := "PREMIXING DB"."MATERIAL SUCTION"."MATERIAL SUCTION BUFF", in2 := 15)
      R_Coil( "PREMIXING DB"."MATERIAL SUCTION"."MATERIAL SUCTION OVER" )
   END_RUNG
   // the same network as SCL:
   IF "AlwaysTRUE" AND ("PREMIXING DB"."MATERIAL SUCTION"."MATERIAL SUCTION BUFF" = 15) AND ("CONTINUE DB"."PREMIXING PROCESS ERROR" <> 1) AND "PREMIXING DB"."MATERIAL SUCTION"."MATERIAL SUCTION OVER" THEN
       "PREMIXING DB"."MATERIAL SUCTION"."MATERIAL SUCTION BUFF" := 0;
   END_IF;
   IF "AlwaysTRUE" AND "PREMIXING DB"."MATERIAL SUCTION"."MATERIAL SUCTION STOP" THEN
       "PREMIXING DB"."MATERIAL SUCTION"."MATERIAL SUCTION BUFF" := 0;
   END_IF;
   IF "PREMIXING DB"."MATERIAL SUCTION"."MATERIAL SUCTION BUFF" <> 15 THEN
       "PREMIXING DB"."MATERIAL SUCTION"."MATERIAL SUCTION OVER" := FALSE;
   END_IF;
END_REGION
END_FUNCTION
